C03701=1106.948,-96.023,-47.577,179.847,4.649,148.823
C03702=1106.943,-95.773,-47.587,179.847,4.654,148.825
C03703=1106.938,-95.524,-47.598,179.847,4.660,148.826
C03704=1106.933,-95.274,-47.609,179.846,4.664,148.827
C03705=1106.927,-95.024,-47.619,179.846,4.669,148.828
C03706=1106.922,-94.775,-47.629,179.846,4.674,148.829
C03707=1106.917,-94.525,-47.640,179.845,4.679,148.830
C03708=1106.911,-94.275,-47.650,179.845,4.684,148.832
C03709=1106.907,-94.025,-47.660,179.844,4.689,148.833
C03710=1106.901,-93.776,-47.670,179.844,4.693,148.834
C03711=1106.896,-93.526,-47.680,179.843,4.698,148.835
C03712=1106.891,-93.276,-47.691,179.843,4.703,148.836
C03713=1106.885,-93.027,-47.702,179.842,4.708,148.838
C03714=1106.880,-92.777,-47.713,179.842,4.713,148.839
C03715=1106.875,-92.527,-47.723,179.842,4.718,148.840
C03716=1106.870,-92.277,-47.733,179.841,4.722,148.841
C03717=1106.864,-92.027,-47.744,179.841,4.728,148.842
C03718=1106.859,-91.778,-47.754,179.841,4.733,148.844
C03719=1106.854,-91.528,-47.765,179.840,4.737,148.845
C03720=1106.848,-91.279,-47.775,179.839,4.743,148.846
C03721=1106.843,-91.028,-47.786,179.839,4.748,148.847
C03722=1106.838,-90.779,-47.796,179.839,4.753,148.849
C03723=1106.833,-90.528,-47.807,179.838,4.757,148.850
C03724=1106.827,-90.280,-47.818,179.838,4.762,148.851
C03725=1106.822,-90.029,-47.828,179.838,4.768,148.852
C03726=1106.817,-89.780,-47.838,179.838,4.773,148.853
C03727=1106.812,-89.530,-47.849,179.837,4.777,148.855
C03728=1106.806,-89.281,-47.860,179.837,4.782,148.856
C03729=1106.801,-89.030,-47.870,179.836,4.787,148.857
C03730=1106.796,-88.781,-47.881,179.836,4.793,148.858
C03731=1106.791,-88.531,-47.891,179.835,4.797,148.860
C03732=1106.786,-88.282,-47.902,179.835,4.802,148.861
C03733=1106.781,-88.031,-47.913,179.835,4.807,148.862
C03734=1106.775,-87.782,-47.923,179.834,4.813,148.863
C03735=1106.770,-87.532,-47.934,179.834,4.817,148.864
C03736=1106.765,-87.283,-47.944,179.833,4.822,148.865
C03737=1106.760,-87.069,-47.953,179.833,4.827,148.867
C03738=1106.756,-86.853,-47.963,179.833,4.831,148.868
C03739=1106.752,-86.640,-47.972,179.833,4.835,148.869
C03740=1106.747,-86.424,-47.981,179.832,4.839,148.870
C03741=1106.742,-86.210,-47.991,179.832,4.844,148.871
C03742=1106.738,-85.995,-47.999,179.832,4.849,148.872
C03743=1106.733,-85.781,-48.009,179.831,4.853,148.873
C03744=1106.729,-85.566,-48.017,179.832,4.857,148.874
C03745=1106.724,-85.316,-48.029,179.831,4.862,148.875
C03746=1106.718,-85.067,-48.039,179.830,4.867,148.876
C03747=1106.714,-84.817,-48.050,179.830,4.872,148.877
C03748=1106.708,-84.568,-48.060,179.830,4.877,148.879
C03749=1106.702,-84.317,-48.072,179.830,4.883,148.880
C03750=1106.698,-84.068,-48.083,179.829,4.888,148.881
C03751=1106.692,-83.818,-48.093,179.829,4.893,148.882
C03752=1106.687,-83.568,-48.104,179.829,4.897,148.883
C03753=1106.682,-83.319,-48.115,179.828,4.902,148.885
C03754=1106.677,-83.069,-48.126,179.828,4.907,148.886
C03755=1106.672,-82.820,-48.136,179.828,4.913,148.887
C03756=1106.666,-82.569,-48.147,179.827,4.918,148.888
C03757=1106.661,-82.320,-48.158,179.827,4.923,148.890
C03758=1106.656,-82.070,-48.169,179.827,4.928,148.891
C03759=1106.651,-81.820,-48.180,179.827,4.934,148.892
C03760=1106.645,-81.571,-48.190,179.827,4.939,148.893
C03761=1106.641,-81.321,-48.201,179.827,4.944,148.894
C03762=1106.634,-81.071,-48.212,179.826,4.948,148.895
C03763=1106.629,-80.822,-48.224,179.826,4.953,148.897
C03764=1106.624,-80.571,-48.234,179.825,4.958,148.898
C03765=1106.619,-80.323,-48.245,179.825,4.964,148.899
C03766=1106.615,-80.073,-48.256,179.825,4.969,148.900
C03767=1106.609,-79.822,-48.268,179.824,4.974,148.902
C03768=1106.603,-79.573,-48.278,179.824,4.979,148.903
C03769=1106.598,-79.323,-48.289,179.824,4.985,148.904
C03770=1106.593,-79.074,-48.300,179.824,4.990,148.905
C03771=1106.587,-78.824,-48.311,179.824,4.995,148.906
C03772=1106.583,-78.574,-48.322,179.824,5.000,148.907
C03773=1106.577,-78.325,-48.333,179.823,5.005,148.909
C03774=1106.572,-78.075,-48.344,179.823,5.010,148.910
C03775=1106.567,-77.825,-48.356,179.823,5.015,148.911
C03776=1106.561,-77.575,-48.366,179.823,5.021,148.912
C03777=1106.557,-77.326,-48.377,179.823,5.026,148.913
C03778=1106.551,-77.077,-48.389,179.823,5.031,148.914
C03779=1106.546,-76.826,-48.399,179.823,5.036,148.916
C03780=1106.541,-76.577,-48.411,179.822,5.041,148.917
C03781=1106.535,-76.327,-48.422,179.822,5.046,148.918
C03782=1106.530,-76.077,-48.433,179.822,5.051,148.919
C03783=1106.525,-75.828,-48.444,179.822,5.057,148.920
C03784=1106.520,-75.578,-48.456,179.822,5.062,148.922
C03785=1106.514,-75.328,-48.466,179.822,5.067,148.923
C03786=1106.510,-75.078,-48.477,179.822,5.072,148.924
C03787=1106.504,-74.829,-48.489,179.821,5.077,148.925
C03788=1106.499,-74.580,-48.500,179.821,5.082,148.926
C03789=1106.494,-74.329,-48.511,179.821,5.087,148.927
C03790=1106.488,-74.079,-48.523,179.821,5.093,148.929
C03791=1106.483,-73.831,-48.534,179.821,5.098,148.930
C03792=1106.478,-73.580,-48.544,179.821,5.103,148.931
C03793=1106.474,-73.365,-48.554,179.820,5.107,148.932
C03794=1106.469,-73.151,-48.564,179.821,5.111,148.933
C03795=1106.465,-72.936,-48.574,179.821,5.115,148.934
C03796=1106.460,-72.722,-48.583,179.820,5.121,148.935
C03797=1106.456,-72.508,-48.593,179.820,5.125,148.936
C03798=1106.451,-72.294,-48.603,179.821,5.129,148.937
C03799=1106.447,-72.079,-48.613,179.820,5.133,148.938
C03800=1106.442,-71.865,-48.622,179.820,5.138,148.939
C03801=1106.437,-71.615,-48.633,179.821,5.143,148.940
C03802=1106.432,-71.365,-48.645,179.820,5.148,148.941
C03803=1106.427,-71.115,-48.657,179.820,5.153,148.942
C03804=1106.422,-70.866,-48.668,179.820,5.159,148.943
C03805=1106.416,-70.616,-48.679,179.820,5.164,148.944
C03806=1106.411,-70.366,-48.690,179.820,5.169,148.946
C03807=1106.406,-70.116,-48.702,179.820,5.174,148.947
C03808=1106.401,-69.867,-48.713,179.820,5.179,148.948
C03809=1106.395,-69.617,-48.725,179.820,5.184,148.949
C03810=1106.390,-69.368,-48.736,179.820,5.189,148.950
C03811=1106.385,-69.118,-48.748,179.820,5.194,148.951
C03812=1106.380,-68.868,-48.759,179.820,5.199,148.952
C03813=1106.374,-68.619,-48.771,179.820,5.204,148.953
C03814=1106.370,-68.369,-48.782,179.820,5.209,148.955
C03815=1106.364,-68.119,-48.794,179.820,5.214,148.956
C03816=1106.359,-67.870,-48.805,179.820,5.219,148.957
C03817=1106.354,-67.620,-48.817,179.820,5.224,148.958
C03818=1106.349,-67.370,-48.828,179.820,5.229,148.959
C03819=1106.343,-67.120,-48.839,179.820,5.234,148.960
C03820=1106.338,-66.871,-48.850,179.821,5.240,148.961
C03821=1106.333,-66.621,-48.862,179.821,5.245,148.962
C03822=1106.328,-66.371,-48.874,179.820,5.250,148.963
C03823=1106.323,-66.121,-48.886,179.821,5.255,148.964
C03824=1106.318,-65.872,-48.898,179.821,5.260,148.965
C03825=1106.312,-65.623,-48.909,179.821,5.265,148.966
C03826=1106.307,-65.373,-48.921,179.821,5.270,148.968
C03827=1106.302,-65.123,-48.932,179.821,5.275,148.969
C03828=1106.297,-64.874,-48.944,179.821,5.280,148.970
C03829=1106.292,-64.624,-48.955,179.821,5.285,148.971
C03830=1106.287,-64.374,-48.967,179.821,5.290,148.972
C03831=1106.281,-64.124,-48.979,179.821,5.295,148.973
C03832=1106.277,-63.874,-48.990,179.822,5.300,148.974
C03833=1106.271,-63.625,-49.002,179.822,5.305,148.975
C03834=1106.266,-63.376,-49.013,179.822,5.310,148.976
C03835=1106.260,-63.126,-49.025,179.822,5.315,148.977
C03836=1106.255,-62.876,-49.038,179.823,5.320,148.978
C03837=1106.251,-62.627,-49.049,179.823,5.325,148.979
C03838=1106.245,-62.377,-49.061,179.823,5.330,148.980
C03839=1106.240,-62.127,-49.073,179.823,5.335,148.981
C03840=1106.235,-61.877,-49.084,179.823,5.340,148.982
C03841=1106.230,-61.627,-49.096,179.823,5.345,148.983
C03842=1106.224,-61.378,-49.109,179.824,5.350,148.984
C03843=1106.220,-61.128,-49.120,179.824,5.355,148.985
C03844=1106.214,-60.878,-49.132,179.824,5.360,148.986
C03845=1106.209,-60.628,-49.144,179.824,5.365,148.987
C03846=1106.204,-60.379,-49.155,179.825,5.369,148.988
C03847=1106.199,-60.130,-49.167,179.825,5.374,148.989
C03848=1106.193,-59.880,-49.179,179.825,5.379,148.990
C03849=1106.189,-59.665,-49.189,179.825,5.383,148.991
C03850=1106.185,-59.451,-49.200,179.825,5.388,148.992
C03851=1106.180,-59.237,-49.209,179.825,5.392,148.993
C03852=1106.176,-59.023,-49.220,179.825,5.396,148.994
C03853=1106.171,-58.808,-49.230,179.825,5.400,148.995
C03854=1106.167,-58.594,-49.241,179.824,5.404,148.996
C03855=1106.162,-58.379,-49.250,179.824,5.408,148.997
C03856=1106.158,-58.165,-49.260,179.824,5.412,148.998
C03857=1106.153,-57.915,-49.273,179.824,5.416,148.999
C03858=1106.148,-57.665,-49.285,179.824,5.421,149.000
C03859=1106.143,-57.416,-49.296,179.824,5.425,149.001
C03860=1106.138,-57.166,-49.309,179.824,5.430,149.002
C03861=1106.132,-56.916,-49.321,179.824,5.436,149.003
C03862=1106.127,-56.667,-49.333,179.824,5.440,149.004
C03863=1106.122,-56.418,-49.345,179.824,5.445,149.005
C03864=1106.117,-56.168,-49.357,179.824,5.449,149.006
C03865=1106.112,-55.918,-49.368,179.823,5.454,149.007
C03866=1106.106,-55.668,-49.381,179.823,5.459,149.008
C03867=1106.101,-55.418,-49.393,179.824,5.464,149.009
C03868=1106.097,-55.169,-49.405,179.823,5.468,149.010
C03869=1106.091,-54.919,-49.417,179.823,5.473,149.012
C03870=1106.086,-54.670,-49.429,179.823,5.478,149.013
C03871=1106.081,-54.420,-49.441,179.823,5.482,149.014
C03872=1106.075,-54.170,-49.453,179.823,5.487,149.015
C03873=1106.070,-53.921,-49.466,179.823,5.492,149.016
C03874=1106.065,-53.671,-49.477,179.822,5.496,149.017
C03875=1106.060,-53.422,-49.490,179.823,5.501,149.018
C03876=1106.055,-53.171,-49.502,179.823,5.506,149.019
C03877=1106.050,-52.922,-49.515,179.822,5.511,149.020
C03878=1106.045,-52.672,-49.526,179.822,5.515,149.021
C03879=1106.040,-52.423,-49.539,179.822,5.520,149.022
C03880=1106.034,-52.173,-49.551,179.822,5.525,149.023
C03881=1106.030,-51.923,-49.562,179.822,5.529,149.024
C03882=1106.025,-51.674,-49.575,179.821,5.534,149.025
C03883=1106.019,-51.425,-49.587,179.821,5.539,149.027
C03884=1106.014,-51.175,-49.599,179.822,5.544,149.028
C03885=1106.009,-50.925,-49.612,179.821,5.548,149.029
C03886=1106.003,-50.675,-49.624,179.821,5.553,149.030
C03887=1105.998,-50.426,-49.636,179.821,5.558,149.031
C03888=1105.993,-50.176,-49.648,179.821,5.562,149.032
C03889=1105.988,-49.926,-49.661,179.821,5.567,149.033
C03890=1105.983,-49.676,-49.673,179.821,5.572,149.034
C03891=1105.978,-49.427,-49.686,179.820,5.576,149.035
C03892=1105.972,-49.177,-49.698,179.820,5.581,149.036
C03893=1105.967,-48.928,-49.710,179.821,5.586,149.037
C03894=1105.962,-48.678,-49.723,179.820,5.591,149.038
C03895=1105.957,-48.428,-49.735,179.820,5.596,149.039
C03896=1105.952,-48.179,-49.747,179.819,5.600,149.041
C03897=1105.947,-47.928,-49.760,179.820,5.605,149.042
C03898=1105.942,-47.679,-49.772,179.820,5.610,149.043
C03899=1105.937,-47.430,-49.785,179.819,5.614,149.044
C03900=1105.931,-47.180,-49.797,179.819,5.619,149.045
C03901=1105.926,-46.931,-49.809,179.819,5.624,149.046
C03902=1105.921,-46.681,-49.822,179.819,5.628,149.047
C03903=1105.915,-46.431,-49.834,179.819,5.633,149.048
C03904=1105.911,-46.181,-49.847,179.819,5.638,149.049
C03905=1105.906,-45.968,-49.857,179.819,5.642,149.050
C03906=1105.902,-45.753,-49.868,179.819,5.646,149.051
C03907=1105.898,-45.539,-49.878,179.818,5.650,149.052
C03908=1105.893,-45.324,-49.889,179.818,5.654,149.053
C03909=1105.889,-45.110,-49.900,179.818,5.658,149.054
C03910=1105.884,-44.896,-49.910,179.817,5.662,149.055
C03911=1105.880,-44.682,-49.921,179.817,5.666,149.056
C03912=1105.876,-44.468,-49.932,179.817,5.670,149.057
C03913=1105.870,-44.218,-49.944,179.817,5.675,149.058
C03914=1105.866,-43.968,-49.957,179.817,5.680,149.059
C03915=1105.861,-43.718,-49.970,179.817,5.684,149.060
C03916=1105.855,-43.468,-49.981,179.817,5.689,149.061
C03917=1105.850,-43.219,-49.994,179.817,5.694,149.062
C03918=1105.845,-42.970,-50.007,179.817,5.698,149.063
C03919=1105.840,-42.720,-50.020,179.816,5.704,149.064
C03920=1105.835,-42.470,-50.033,179.817,5.708,149.065
C03921=1105.829,-42.220,-50.045,179.817,5.713,149.066
C03922=1105.824,-41.971,-50.057,179.817,5.718,149.067
C03923=1105.819,-41.721,-50.070,179.818,5.723,149.068
C03924=1105.814,-41.471,-50.083,179.818,5.728,149.069
C03925=1105.809,-41.222,-50.096,179.818,5.733,149.070
C03926=1105.804,-40.972,-50.107,179.819,5.738,149.071
C03927=1105.799,-40.723,-50.120,179.819,5.742,149.072
C03928=1105.793,-40.473,-50.134,179.819,5.747,149.073
C03929=1105.788,-40.223,-50.146,179.819,5.752,149.074
C03930=1105.783,-39.974,-50.159,179.820,5.757,149.075
C03931=1105.778,-39.725,-50.171,179.820,5.762,149.076
C03932=1105.774,-39.475,-50.184,179.821,5.766,149.077
C03933=1105.768,-39.225,-50.197,179.821,5.770,149.078
C03934=1105.762,-38.975,-50.209,179.821,5.775,149.079
C03935=1105.757,-38.726,-50.222,179.821,5.780,149.080
C03936=1105.753,-38.476,-50.235,179.821,5.785,149.081
C03937=1105.747,-38.226,-50.248,179.822,5.790,149.082
C03938=1105.742,-37.977,-50.260,179.822,5.794,149.083
C03939=1105.737,-37.727,-50.274,179.822,5.798,149.083
C03940=1105.732,-37.477,-50.286,179.823,5.803,149.084
C03941=1105.727,-37.228,-50.299,179.823,5.808,149.085
C03942=1105.722,-36.979,-50.312,179.823,5.812,149.086
C03943=1105.716,-36.728,-50.325,179.824,5.817,149.087
C03944=1105.711,-36.479,-50.338,179.824,5.821,149.088
C03945=1105.706,-36.230,-50.350,179.825,5.825,149.089
C03946=1105.702,-35.980,-50.363,179.825,5.830,149.090
C03947=1105.696,-35.730,-50.376,179.826,5.835,149.091
C03948=1105.691,-35.481,-50.389,179.825,5.839,149.091
C03949=1105.686,-35.231,-50.402,179.826,5.844,149.092
C03950=1105.680,-34.981,-50.415,179.826,5.848,149.093
C03951=1105.675,-34.732,-50.428,179.827,5.853,149.094
C03952=1105.671,-34.482,-50.441,179.827,5.857,149.095
C03953=1105.666,-34.233,-50.453,179.827,5.862,149.096
C03954=1105.660,-33.984,-50.467,179.828,5.866,149.097
C03955=1105.655,-33.733,-50.480,179.828,5.870,149.098
C03956=1105.650,-33.484,-50.493,179.828,5.875,149.098
C03957=1105.645,-33.234,-50.506,179.829,5.880,149.099
C03958=1105.640,-32.985,-50.519,179.829,5.883,149.100
C03959=1105.635,-32.735,-50.532,179.829,5.888,149.101
C03960=1105.630,-32.485,-50.545,179.830,5.893,149.102
C03961=1105.626,-32.271,-50.556,179.830,5.896,149.103
C03962=1105.621,-32.057,-50.568,179.830,5.900,149.104
C03963=1105.617,-31.842,-50.579,179.830,5.904,149.104
C03964=1105.612,-31.628,-50.590,179.830,5.907,149.105
C03965=1105.607,-31.413,-50.601,179.831,5.912,149.106
C03966=1105.603,-31.200,-50.612,179.831,5.916,149.107
C03967=1105.598,-30.986,-50.624,179.832,5.919,149.107
C03968=1105.594,-30.772,-50.634,179.831,5.923,149.108
C03969=1105.589,-30.522,-50.649,179.832,5.928,149.109
C03970=1105.584,-30.273,-50.661,179.832,5.932,149.110
C03971=1105.580,-30.023,-50.674,179.832,5.937,149.111
C03972=1105.574,-29.773,-50.687,179.833,5.941,149.112
C03973=1105.569,-29.523,-50.700,179.833,5.945,149.113
C03974=1105.564,-29.274,-50.714,179.833,5.950,149.114
C03975=1105.559,-29.025,-50.727,179.834,5.955,149.115
C03976=1105.554,-28.775,-50.740,179.833,5.959,149.116
C03977=1105.548,-28.525,-50.753,179.834,5.963,149.116
C03978=1105.544,-28.276,-50.767,179.834,5.968,149.117
C03979=1105.538,-28.026,-50.780,179.834,5.972,149.118
C03980=1105.534,-27.776,-50.793,179.835,5.977,149.119
C03981=1105.528,-27.527,-50.807,179.835,5.982,149.120
C03982=1105.524,-27.277,-50.820,179.835,5.985,149.121
C03983=1105.518,-27.027,-50.833,179.835,5.991,149.122
C03984=1105.514,-26.778,-50.847,179.835,5.995,149.123
C03985=1105.508,-26.528,-50.860,179.835,5.999,149.124
C03986=1105.503,-26.278,-50.873,179.836,6.004,149.125
C03987=1105.498,-26.029,-50.887,179.836,6.009,149.126
C03988=1105.493,-25.779,-50.900,179.836,6.014,149.127
C03989=1105.487,-25.530,-50.913,179.836,6.018,149.128
C03990=1105.483,-25.280,-50.927,179.837,6.022,149.129
C03991=1105.477,-25.031,-50.940,179.837,6.028,149.130
C03992=1105.473,-24.781,-50.953,179.837,6.032,149.131
C03993=1105.467,-24.532,-50.967,179.837,6.037,149.132
C03994=1105.463,-24.282,-50.980,179.838,6.042,149.133
C03995=1105.457,-24.033,-50.994,179.838,6.046,149.133
C03996=1105.452,-23.782,-51.007,179.838,6.051,149.135
C03997=1105.447,-23.533,-51.020,179.838,6.056,149.135
C03998=1105.442,-23.283,-51.034,179.839,6.060,149.136
C03999=1105.437,-23.034,-51.047,179.839,6.065,149.137
C04000=1105.432,-22.784,-51.061,179.840,6.070,149.138
C04001=1105.426,-22.535,-51.073,179.840,6.074,149.139
C04002=1105.421,-22.285,-51.088,179.840,6.078,149.140
C04003=1105.416,-22.036,-51.100,179.840,6.083,149.141
C04004=1105.411,-21.786,-51.115,179.841,6.088,149.142
C04005=1105.406,-21.536,-51.128,179.841,6.093,149.143
C04006=1105.401,-21.287,-51.142,179.842,6.098,149.144
C04007=1105.395,-21.037,-51.155,179.841,6.102,149.145
C04008=1105.391,-20.788,-51.169,179.842,6.106,149.146
C04009=1105.386,-20.538,-51.183,179.842,6.111,149.147
C04010=1105.380,-20.289,-51.196,179.843,6.116,149.147
C04011=1105.375,-20.039,-51.210,179.843,6.120,149.148
C04012=1105.370,-19.790,-51.223,179.844,6.125,149.149
C04013=1105.365,-19.540,-51.237,179.844,6.129,149.150
C04014=1105.360,-19.290,-51.251,179.844,6.134,149.151
C04015=1105.355,-19.041,-51.264,179.845,6.139,149.152
C04016=1105.350,-18.791,-51.278,179.845,6.143,149.153
C04017=1105.346,-18.577,-51.289,179.845,6.147,149.154
C04018=1105.341,-18.363,-51.302,179.846,6.152,149.154
C04019=1105.337,-18.149,-51.313,179.846,6.155,149.155
C04020=1105.333,-17.935,-51.324,179.846,6.159,149.156
C04021=1105.328,-17.721,-51.336,179.847,6.163,149.157
C04022=1105.324,-17.507,-51.348,179.847,6.167,149.158
C04023=1105.320,-17.292,-51.361,179.847,6.171,149.158
C04024=1105.315,-17.078,-51.372,179.848,6.174,149.159
C04025=1105.310,-16.829,-51.385,179.848,6.179,149.160
C04026=1105.305,-16.579,-51.400,179.849,6.184,149.161
C04027=1105.300,-16.329,-51.413,179.849,6.189,149.162
C04028=1105.295,-16.080,-51.427,179.850,6.193,149.163
C04029=1105.290,-15.830,-51.441,179.850,6.197,149.163
C04030=1105.285,-15.580,-51.454,179.850,6.202,149.164
C04031=1105.279,-15.331,-51.468,179.851,6.207,149.165
C04032=1105.275,-15.081,-51.483,179.851,6.211,149.166
C04033=1105.270,-14.832,-51.496,179.852,6.216,149.167
C04034=1105.264,-14.582,-51.509,179.853,6.220,149.168
C04035=1105.259,-14.333,-51.524,179.853,6.224,149.169
C04036=1105.255,-14.083,-51.538,179.853,6.229,149.169
C04037=1105.250,-13.834,-51.551,179.854,6.234,149.170
C04038=1105.245,-13.584,-51.566,179.854,6.239,149.171
C04039=1105.239,-13.334,-51.579,179.855,6.243,149.172
C04040=1105.234,-13.085,-51.593,179.856,6.248,149.173
C04041=1105.229,-12.835,-51.607,179.855,6.251,149.174
C04042=1105.224,-12.586,-51.622,179.856,6.256,149.175
C04043=1105.220,-12.336,-51.635,179.856,6.261,149.176
C04044=1105.214,-12.087,-51.649,179.857,6.266,149.176
C04045=1105.209,-11.837,-51.663,179.857,6.270,149.177
C04046=1105.204,-11.587,-51.677,179.858,6.275,149.178
C04047=1105.199,-11.338,-51.691,179.858,6.279,149.179
C04048=1105.194,-11.089,-51.705,179.859,6.283,149.180
C04049=1105.189,-10.839,-51.719,179.859,6.288,149.181
C04050=1105.184,-10.589,-51.733,179.860,6.293,149.182
C04051=1105.179,-10.340,-51.747,179.861,6.297,149.182
C04052=1105.174,-10.091,-51.761,179.861,6.302,149.183
C04053=1105.169,-9.841,-51.776,179.862,6.307,149.184
C04054=1105.164,-9.591,-51.790,179.862,6.310,149.185
C04055=1105.159,-9.342,-51.804,179.862,6.315,149.186
C04056=1105.153,-9.093,-51.818,179.863,6.320,149.187
C04057=1105.148,-8.842,-51.832,179.864,6.324,149.187
C04058=1105.143,-8.593,-51.846,179.864,6.329,149.188
C04059=1105.138,-8.343,-51.860,179.865,6.334,149.189
C04060=1105.133,-8.094,-51.874,179.866,6.338,149.190
C04061=1105.128,-7.844,-51.888,179.866,6.342,149.191
C04062=1105.123,-7.594,-51.903,179.866,6.347,149.192
C04063=1105.118,-7.345,-51.918,179.867,6.351,149.193
C04064=1105.113,-7.096,-51.932,179.868,6.356,149.193
C04065=1105.108,-6.847,-51.946,179.868,6.360,149.194
C04066=1105.103,-6.597,-51.960,179.869,6.365,149.195
C04067=1105.098,-6.347,-51.974,179.869,6.370,149.196
C04068=1105.093,-6.097,-51.989,179.870,6.373,149.197
C04069=1105.088,-5.848,-52.003,179.870,6.378,149.198
C04070=1105.083,-5.598,-52.017,179.871,6.383,149.198
C04071=1105.077,-5.349,-52.031,179.872,6.387,149.199
C04072=1105.072,-5.099,-52.045,179.872,6.392,149.200
C04073=1105.068,-4.885,-52.058,179.873,6.395,149.201
C04074=1105.064,-4.671,-52.070,179.873,6.400,149.202
C04075=1105.060,-4.457,-52.083,179.873,6.404,149.202
C04076=1105.055,-4.243,-52.095,179.874,6.407,149.203
C04077=1105.052,-4.029,-52.107,179.875,6.412,149.204
C04078=1105.047,-3.815,-52.119,179.875,6.415,149.204
C04079=1105.043,-3.601,-52.131,179.875,6.419,149.205
C04080=1105.038,-3.386,-52.144,179.876,6.423,149.206
C04081=1105.033,-3.138,-52.159,179.877,6.428,149.206
C04082=1105.028,-2.888,-52.173,179.877,6.432,149.207
C04083=1105.023,-2.638,-52.187,179.878,6.436,149.208
C04084=1105.018,-2.389,-52.202,179.878,6.441,149.209
C04085=1105.013,-2.139,-52.217,179.879,6.445,149.210
C04086=1105.008,-1.890,-52.231,179.880,6.450,149.211
C04087=1105.003,-1.640,-52.245,179.880,6.455,149.212
C04088=1104.998,-1.390,-52.259,179.881,6.459,149.212
C04089=1104.993,-1.140,-52.274,179.882,6.464,149.213
C04090=1104.987,-0.892,-52.289,179.882,6.468,149.214
C04091=1104.982,-0.642,-52.303,179.883,6.473,149.215
C04092=1104.978,-0.392,-52.317,179.884,6.478,149.216
C04093=1104.973,-0.143,-52.332,179.884,6.481,149.216
C04094=1104.968,0.106,-52.347,179.884,6.486,149.217
C04095=1104.963,0.356,-52.361,179.885,6.490,149.218
C04096=1104.958,0.605,-52.377,179.886,6.495,149.219
C04097=1104.953,0.855,-52.391,179.886,6.500,149.220
C04098=1104.948,1.105,-52.405,179.887,6.504,149.220
C04099=1104.943,1.354,-52.420,179.888,6.509,149.221
C04100=1104.938,1.604,-52.434,179.888,6.514,149.222
C04101=1104.932,1.854,-52.449,179.889,6.518,149.223
C04102=1104.928,2.103,-52.464,179.890,6.523,149.224
C04103=1104.923,2.352,-52.479,179.890,6.527,149.225
C04104=1104.918,2.602,-52.494,179.891,6.532,149.226
C04105=1104.912,2.852,-52.508,179.892,6.536,149.226
C04106=1104.907,3.101,-52.523,179.892,6.541,149.227
C04107=1104.903,3.350,-52.538,179.893,6.546,149.228
C04108=1104.898,3.600,-52.552,179.893,6.551,149.229
C04109=1104.892,3.850,-52.568,179.894,6.555,149.230
C04110=1104.888,4.099,-52.582,179.895,6.560,149.231
C04111=1104.883,4.348,-52.597,179.896,6.564,149.231
C04112=1104.878,4.598,-52.611,179.896,6.569,149.232
C04113=1104.873,4.847,-52.627,179.897,6.573,149.233
C04114=1104.868,5.097,-52.641,179.898,6.578,149.234
C04115=1104.863,5.346,-52.656,179.898,6.583,149.235
C04116=1104.857,5.596,-52.671,179.899,6.587,149.235
C04117=1104.853,5.845,-52.686,179.900,6.592,149.236
C04118=1104.848,6.095,-52.700,179.900,6.596,149.237
C04119=1104.842,6.344,-52.716,179.901,6.601,149.238
C04120=1104.837,6.594,-52.730,179.902,6.606,149.239
C04121=1104.833,6.843,-52.745,179.902,6.610,149.240
C04122=1104.827,7.093,-52.761,179.903,6.615,149.241
C04123=1104.822,7.342,-52.775,179.903,6.620,149.241
C04124=1104.818,7.591,-52.790,179.904,6.624,149.242
C04125=1104.812,7.841,-52.805,179.905,6.629,149.243
C04126=1104.807,8.091,-52.820,179.906,6.633,149.244
C04127=1104.803,8.341,-52.836,179.906,6.638,149.245
C04128=1104.798,8.590,-52.850,179.907,6.643,149.246
C04129=1104.793,8.804,-52.863,179.907,6.646,149.246
C04130=1104.789,9.019,-52.876,179.907,6.650,149.247
C04131=1104.785,9.232,-52.888,179.908,6.655,149.248
C04132=1104.780,9.446,-52.902,179.908,6.658,149.248
C04133=1104.776,9.660,-52.914,179.908,6.662,149.249
C04134=1104.771,9.874,-52.927,179.909,6.666,149.250
C04135=1104.767,10.088,-52.941,179.909,6.669,149.251
C04136=1104.763,10.302,-52.953,179.909,6.673,149.252
C04137=1104.758,10.551,-52.968,179.910,6.678,149.252
C04138=1104.754,10.801,-52.984,179.910,6.682,149.253
C04139=1104.748,11.050,-52.999,179.910,6.686,149.254
C04140=1104.743,11.300,-53.013,179.911,6.691,149.255
C04141=1104.738,11.549,-53.029,179.911,6.696,149.256
C04142=1104.733,11.799,-53.044,179.912,6.700,149.257
C04143=1104.728,12.048,-53.060,179.912,6.704,149.258
C04144=1104.723,12.298,-53.074,179.913,6.709,149.258
C04145=1104.718,12.548,-53.090,179.913,6.713,149.259
C04146=1104.713,12.797,-53.105,179.913,6.717,149.260
C04147=1104.708,13.046,-53.120,179.914,6.722,149.261
C04148=1104.703,13.296,-53.135,179.914,6.727,149.262
C04149=1104.698,13.545,-53.150,179.914,6.731,149.263
C04150=1104.693,13.794,-53.165,179.915,6.735,149.264
C04151=1104.688,14.044,-53.181,179.916,6.740,149.264
C04152=1104.684,14.294,-53.196,179.916,6.743,149.265
C04153=1104.678,14.543,-53.212,179.916,6.748,149.266
C04154=1104.674,14.792,-53.227,179.917,6.753,149.267
C04155=1104.668,15.042,-53.242,179.917,6.756,149.268
C04156=1104.663,15.291,-53.257,179.918,6.761,149.269
C04157=1104.658,15.541,-53.273,179.919,6.766,149.270
C04158=1104.653,15.791,-53.288,179.919,6.771,149.270
C04159=1104.648,16.040,-53.303,179.920,6.774,149.271
C04160=1104.643,16.289,-53.319,179.920,6.779,149.272
C04161=1104.638,16.538,-53.334,179.921,6.783,149.273
C04162=1104.634,16.788,-53.350,179.921,6.787,149.274
C04163=1104.628,17.038,-53.365,179.922,6.792,149.274
C04164=1104.624,17.287,-53.380,179.922,6.796,149.275
C04165=1104.618,17.536,-53.396,179.922,6.800,149.276
C04166=1104.614,17.787,-53.411,179.923,6.805,149.277
C04167=1104.608,18.036,-53.426,179.924,6.809,149.278
C04168=1104.603,18.286,-53.442,179.924,6.813,149.279
C04169=1104.598,18.535,-53.457,179.925,6.818,149.279
C04170=1104.594,18.785,-53.473,179.925,6.822,149.280
C04171=1104.588,19.034,-53.488,179.926,6.826,149.281
C04172=1104.584,19.283,-53.503,179.926,6.830,149.282
C04173=1104.578,19.533,-53.519,179.927,6.835,149.283
C04174=1104.574,19.782,-53.535,179.927,6.839,149.283
C04175=1104.569,20.031,-53.550,179.928,6.843,149.284
C04176=1104.564,20.281,-53.566,179.929,6.848,149.285
C04177=1104.558,20.530,-53.582,179.929,6.852,149.286
C04178=1104.554,20.780,-53.597,179.929,6.856,149.287
C04179=1104.549,21.029,-53.613,179.930,6.861,149.287
C04180=1104.543,21.279,-53.628,179.930,6.865,149.288
C04181=1104.539,21.529,-53.644,179.931,6.869,149.289
C04182=1104.534,21.778,-53.659,179.932,6.874,149.290
C04183=1104.529,22.027,-53.675,179.933,6.878,149.290
C04184=1104.524,22.277,-53.691,179.933,6.882,149.291
C04185=1104.520,22.491,-53.703,179.933,6.885,149.292
C04186=1104.516,22.704,-53.718,179.934,6.889,149.293
C04187=1104.511,22.918,-53.731,179.935,6.893,149.293
C04188=1104.506,23.132,-53.745,179.935,6.897,149.294
C04189=1104.503,23.346,-53.758,179.936,6.900,149.294
C04190=1104.498,23.560,-53.771,179.936,6.904,149.295
C04191=1104.494,23.774,-53.785,179.937,6.907,149.296
C04192=1104.490,23.988,-53.798,179.937,6.911,149.296
C04193=1104.485,24.238,-53.814,179.938,6.915,149.297
C04194=1104.480,24.486,-53.830,179.939,6.920,149.298
C04195=1104.475,24.737,-53.846,179.939,6.923,149.299
C04196=1104.470,24.986,-53.861,179.940,6.928,149.299
C04197=1104.465,25.235,-53.877,179.941,6.932,149.300
C04198=1104.460,25.485,-53.893,179.941,6.936,149.301
C04199=1104.455,25.734,-53.909,179.942,6.940,149.302
C04200=1104.450,25.983,-53.924,179.943,6.945,149.302
C04201=1104.445,26.233,-53.940,179.943,6.948,149.303
C04202=1104.441,26.482,-53.956,179.944,6.953,149.304
C04203=1104.435,26.731,-53.972,179.945,6.957,149.305
C04204=1104.430,26.981,-53.988,179.945,6.961,149.305
C04205=1104.425,27.231,-54.003,179.946,6.966,149.306
C04206=1104.420,27.480,-54.020,179.947,6.970,149.307
C04207=1104.415,27.730,-54.035,179.948,6.974,149.307
C04208=1104.410,27.979,-54.051,179.948,6.978,149.308
C04209=1104.405,28.229,-54.068,179.949,6.982,149.309
C04210=1104.401,28.478,-54.083,179.950,6.987,149.310
C04211=1104.396,28.728,-54.099,179.950,6.991,149.311
C04212=1104.391,28.977,-54.115,179.951,6.995,149.311
C04213=1104.386,29.227,-54.131,179.952,6.999,149.312
C04214=1104.381,29.475,-54.147,179.953,7.003,149.313
C04215=1104.375,29.725,-54.163,179.953,7.007,149.313
C04216=1104.371,29.975,-54.179,179.954,7.012,149.314
C04217=1104.366,30.224,-54.195,179.955,7.015,149.315
C04218=1104.361,30.474,-54.211,179.956,7.020,149.315
C04219=1104.356,30.723,-54.227,179.956,7.024,149.316
C04220=1104.351,30.973,-54.243,179.957,7.028,149.317
C04221=1104.346,31.221,-54.260,179.958,7.032,149.318
C04222=1104.341,31.472,-54.276,179.959,7.036,149.318
C04223=1104.336,31.720,-54.292,179.959,7.040,149.319
C04224=1104.331,31.970,-54.308,179.960,7.045,149.320
C04225=1104.326,32.220,-54.323,179.961,7.049,149.320
C04226=1104.321,32.469,-54.340,179.962,7.052,149.321
C04227=1104.316,32.719,-54.356,179.963,7.057,149.322
C04228=1104.311,32.968,-54.372,179.964,7.061,149.322
C04229=1104.306,33.217,-54.389,179.964,7.065,149.323
C04230=1104.301,33.466,-54.404,179.965,7.069,149.324
C04231=1104.297,33.716,-54.421,179.966,7.074,149.325
C04232=1104.291,33.965,-54.436,179.966,7.077,149.325
C04233=1104.287,34.215,-54.453,179.967,7.081,149.326
C04234=1104.282,34.465,-54.469,179.968,7.086,149.327
C04235=1104.277,34.714,-54.485,179.969,7.090,149.327
C04236=1104.272,34.964,-54.501,179.970,7.093,149.328
C04237=1104.267,35.213,-54.518,179.970,7.098,149.329
C04238=1104.262,35.462,-54.534,179.971,7.102,149.329
C04239=1104.257,35.711,-54.550,179.972,7.106,149.330
C04240=1104.253,35.961,-54.567,179.973,7.110,149.331
C04241=1104.248,36.175,-54.580,179.974,7.113,149.331
C04242=1104.244,36.388,-54.594,179.974,7.117,149.332
C04243=1104.240,36.602,-54.609,179.975,7.120,149.332
C04244=1104.235,36.816,-54.622,179.976,7.124,149.333
C04245=1104.231,37.029,-54.637,179.977,7.128,149.334
C04246=1104.227,37.244,-54.650,179.977,7.131,149.334
C04247=1104.223,37.457,-54.665,179.978,7.135,149.335
C04248=1104.218,37.672,-54.678,179.979,7.138,149.335
C04249=1104.213,37.920,-54.695,179.980,7.142,149.336
C04250=1104.208,38.170,-54.712,179.981,7.147,149.337
C04251=1104.203,38.420,-54.729,179.981,7.150,149.337
C04252=1104.198,38.669,-54.744,179.982,7.154,149.338
C04253=1104.194,38.919,-54.761,179.983,7.159,149.339
C04254=1104.189,39.167,-54.777,179.984,7.162,149.339
C04255=1104.184,39.417,-54.794,179.985,7.167,149.340
C04256=1104.179,39.667,-54.810,179.986,7.171,149.341
C04257=1104.173,39.916,-54.827,179.986,7.174,149.341
C04258=1104.169,40.166,-54.843,179.987,7.179,149.342
C04259=1104.164,40.414,-54.860,179.989,7.183,149.343
C04260=1104.159,40.664,-54.876,179.990,7.187,149.343
C04261=1104.154,40.914,-54.893,179.991,7.190,149.344
C04262=1104.149,41.163,-54.909,179.992,7.195,149.344
C04263=1104.144,41.412,-54.926,179.993,7.199,149.345
C04264=1104.140,41.662,-54.943,179.993,7.203,149.346
C04265=1104.134,41.911,-54.959,179.994,7.207,149.346
C04266=1104.130,42.161,-54.976,179.995,7.211,149.347
C04267=1104.124,42.410,-54.992,179.996,7.215,149.348
C04268=1104.120,42.659,-55.008,179.997,7.219,149.348
C04269=1104.114,42.909,-55.026,179.998,7.223,149.349
C04270=1104.109,43.158,-55.042,179.999,7.228,149.350
C04271=1104.105,43.407,-55.059,180.000,7.231,149.350
C04272=1104.100,43.657,-55.076,-179.999,7.235,149.351
C04273=1104.095,43.906,-55.092,-179.998,7.239,149.351
C04274=1104.090,44.156,-55.109,-179.997,7.243,149.352
C04275=1104.086,44.405,-55.125,-179.996,7.247,149.353
C04276=1104.080,44.655,-55.143,-179.995,7.251,149.353
C04277=1104.075,44.904,-55.159,-179.995,7.255,149.354
C04278=1104.071,45.153,-55.176,-179.993,7.259,149.354
C04279=1104.066,45.403,-55.193,-179.992,7.263,149.355
C04280=1104.061,45.652,-55.209,-179.991,7.267,149.356
C04281=1104.056,45.901,-55.226,-179.991,7.271,149.356
C04282=1104.051,46.151,-55.243,-179.990,7.275,149.357
C04283=1104.046,46.400,-55.260,-179.988,7.279,149.357
C04284=1104.041,46.650,-55.277,-179.988,7.283,149.358
C04285=1104.036,46.899,-55.293,-179.987,7.287,149.359
C04286=1104.032,47.148,-55.310,-179.985,7.291,149.359
C04287=1104.026,47.398,-55.327,-179.984,7.296,149.360
C04288=1104.021,47.647,-55.344,-179.983,7.299,149.360
C04289=1104.016,47.897,-55.361,-179.982,7.303,149.361
C04290=1104.012,48.146,-55.378,-179.981,7.307,149.362
C04291=1104.007,48.396,-55.394,-179.981,7.311,149.362
C04292=1104.002,48.644,-55.412,-179.979,7.315,149.363
C04293=1103.997,48.894,-55.429,-179.978,7.319,149.364
C04294=1103.992,49.144,-55.446,-179.977,7.323,149.364
C04295=1103.987,49.393,-55.463,-179.977,7.327,149.365
C04296=1103.982,49.642,-55.479,-179.975,7.331,149.365
C04297=1103.978,49.856,-55.494,-179.975,7.334,149.366
C04298=1103.974,50.070,-55.508,-179.973,7.338,149.366
C04299=1103.970,50.283,-55.523,-179.972,7.341,149.367
C04300=1103.966,50.497,-55.537,-179.972,7.345,149.367
C04301=1103.961,50.711,-55.552,-179.971,7.348,149.368
C04302=1103.957,50.925,-55.567,-179.970,7.351,149.368
C04303=1103.953,51.138,-55.582,-179.969,7.355,149.369
C04304=1103.949,51.352,-55.597,-179.968,7.358,149.369
C04305=1103.944,51.601,-55.613,-179.967,7.362,149.370
C04306=1103.939,51.851,-55.631,-179.966,7.366,149.371
C04307=1103.934,52.100,-55.647,-179.965,7.370,149.371
C04308=1103.929,52.349,-55.665,-179.964,7.374,149.372
C04309=1103.924,52.598,-55.682,-179.963,7.378,149.372
C04310=1103.919,52.848,-55.699,-179.962,7.382,149.373
C04311=1103.915,53.098,-55.716,-179.960,7.386,149.373
C04312=1103.910,53.347,-55.734,-179.959,7.390,149.374
C04313=1103.905,53.596,-55.750,-179.958,7.394,149.375
C04314=1103.899,53.846,-55.767,-179.957,7.398,149.375
C04315=1103.895,54.095,-55.785,-179.956,7.402,149.376
C04316=1103.890,54.344,-55.802,-179.955,7.406,149.376
C04317=1103.885,54.594,-55.819,-179.954,7.409,149.377
C04318=1103.881,54.843,-55.836,-179.953,7.414,149.377
C04319=1103.875,55.093,-55.854,-179.951,7.417,149.378
C04320=1103.871,55.342,-55.872,-179.950,7.422,149.379
C04321=1103.865,55.591,-55.888,-179.950,7.425,149.379
C04322=1103.860,55.840,-55.905,-179.948,7.429,149.380
C04323=1103.855,56.090,-55.923,-179.947,7.433,149.380
C04324=1103.851,56.339,-55.940,-179.945,7.437,149.381
C04325=1103.846,56.588,-55.958,-179.945,7.441,149.381
C04326=1103.841,56.838,-55.975,-179.944,7.445,149.382
C04327=1103.837,57.087,-55.992,-179.942,7.449,149.383
C04328=1103.831,57.337,-56.010,-179.941,7.453,149.383
C04329=1103.826,57.586,-56.027,-179.940,7.457,149.384
C04330=1103.822,57.835,-56.044,-179.939,7.461,149.384
C04331=1103.817,58.085,-56.062,-179.938,7.465,149.385
C04332=1103.812,58.334,-56.080,-179.936,7.469,149.385
C04333=1103.808,58.583,-56.097,-179.935,7.473,149.386
C04334=1103.802,58.832,-56.114,-179.934,7.476,149.386
C04335=1103.797,59.081,-56.132,-179.933,7.481,149.387
C04336=1103.792,59.331,-56.149,-179.932,7.485,149.388
C04337=1103.788,59.580,-56.167,-179.931,7.489,149.388
C04338=1103.782,59.830,-56.184,-179.930,7.492,149.389
C04339=1103.777,60.079,-56.202,-179.929,7.496,149.389
C04340=1103.773,60.329,-56.218,-179.927,7.500,149.390
C04341=1103.768,60.578,-56.236,-179.926,7.504,149.390
C04342=1103.763,60.827,-56.254,-179.924,7.508,149.391
C04343=1103.758,61.077,-56.272,-179.924,7.512,149.391
C04344=1103.753,61.326,-56.290,-179.922,7.516,149.392
C04345=1103.749,61.575,-56.307,-179.921,7.520,149.393
C04346=1103.744,61.825,-56.324,-179.920,7.524,149.393
C04347=1103.739,62.074,-56.342,-179.919,7.528,149.394
C04348=1103.734,62.323,-56.360,-179.918,7.531,149.394
C04349=1103.729,62.573,-56.378,-179.916,7.535,149.394
C04350=1103.724,62.822,-56.395,-179.915,7.540,149.395
C04351=1103.719,63.071,-56.413,-179.913,7.543,149.396
C04352=1103.714,63.321,-56.430,-179.912,7.548,149.396
C04353=1103.710,63.535,-56.446,-179.911,7.551,149.397
C04354=1103.706,63.748,-56.461,-179.910,7.554,149.397
C04355=1103.702,63.962,-56.476,-179.909,7.557,149.398
C04356=1103.698,64.175,-56.491,-179.908,7.561,149.398
C04357=1103.694,64.389,-56.507,-179.907,7.564,149.398
C04358=1103.690,64.602,-56.522,-179.906,7.567,149.399
C04359=1103.685,64.816,-56.537,-179.906,7.571,149.400
C04360=1103.681,65.029,-56.552,-179.904,7.575,149.400
C04361=1103.677,65.279,-56.570,-179.902,7.579,149.400
C04362=1103.672,65.529,-56.587,-179.901,7.582,149.401
C04363=1103.667,65.778,-56.605,-179.900,7.586,149.401
C04364=1103.662,66.027,-56.623,-179.899,7.590,149.402
C04365=1103.657,66.276,-56.641,-179.898,7.594,149.403
C04366=1103.652,66.525,-56.659,-179.896,7.598,149.403
C04367=1103.647,66.774,-56.677,-179.895,7.601,149.403
C04368=1103.642,67.024,-56.695,-179.894,7.606,149.404
C04369=1103.637,67.273,-56.713,-179.892,7.609,149.405
C04370=1103.632,67.523,-56.731,-179.891,7.614,149.405
C04371=1103.628,67.773,-56.749,-179.890,7.618,149.406
C04372=1103.623,68.022,-56.767,-179.888,7.622,149.406
C04373=1103.618,68.271,-56.785,-179.888,7.625,149.407
C04374=1103.613,68.520,-56.803,-179.886,7.629,149.407
C04375=1103.608,68.769,-56.821,-179.885,7.633,149.408
C04376=1103.603,69.018,-56.839,-179.883,7.637,149.408
C04377=1103.599,69.268,-56.857,-179.882,7.641,149.409
C04378=1103.594,69.517,-56.875,-179.881,7.645,149.409
C04379=1103.589,69.767,-56.893,-179.879,7.649,149.410
C04380=1103.584,70.016,-56.911,-179.878,7.652,149.410
C04381=1103.580,70.265,-56.929,-179.877,7.657,149.411
C04382=1103.575,70.514,-56.947,-179.876,7.660,149.411
C04383=1103.570,70.763,-56.965,-179.874,7.664,149.412
C04384=1103.565,71.013,-56.983,-179.873,7.669,149.412
C04385=1103.560,71.262,-57.001,-179.871,7.673,149.413
C04386=1103.556,71.512,-57.019,-179.870,7.676,149.413
C04387=1103.551,71.761,-57.037,-179.869,7.680,149.414
C04388=1103.546,72.010,-57.055,-179.868,7.684,149.414
C04389=1103.541,72.259,-57.073,-179.866,7.688,149.415
C04390=1103.537,72.509,-57.092,-179.865,7.692,149.415
C04391=1103.531,72.758,-57.110,-179.863,7.696,149.416
C04392=1103.526,73.008,-57.128,-179.862,7.700,149.416
C04393=1103.521,73.256,-57.147,-179.861,7.704,149.417
C04394=1103.517,73.506,-57.165,-179.859,7.708,149.417
C04395=1103.512,73.755,-57.183,-179.858,7.711,149.418
C04396=1103.507,74.004,-57.201,-179.857,7.715,149.418
C04397=1103.502,74.254,-57.219,-179.856,7.719,149.419
C04398=1103.498,74.503,-57.238,-179.854,7.723,149.419
C04399=1103.493,74.752,-57.257,-179.853,7.728,149.420
C04400=1103.488,75.002,-57.275,-179.851,7.731,149.420
C04401=1103.483,75.251,-57.293,-179.850,7.735,149.421
C04402=1103.479,75.501,-57.311,-179.849,7.740,149.422
C04403=1103.474,75.749,-57.330,-179.847,7.743,149.422
C04404=1103.468,75.999,-57.348,-179.846,7.747,149.422
C04405=1103.463,76.248,-57.366,-179.844,7.751,149.423
C04406=1103.459,76.498,-57.385,-179.843,7.755,149.423
C04407=1103.454,76.746,-57.403,-179.842,7.759,149.424
C04408=1103.449,76.996,-57.422,-179.840,7.763,149.424
C04409=1103.446,77.209,-57.438,-179.839,7.766,149.425
C04410=1103.441,77.423,-57.453,-179.839,7.769,149.425
C04411=1103.437,77.636,-57.469,-179.838,7.772,149.426
C04412=1103.433,77.850,-57.485,-179.837,7.775,149.426
C04413=1103.429,78.064,-57.501,-179.836,7.779,149.427
C04414=1103.424,78.277,-57.517,-179.835,7.782,149.427
C04415=1103.420,78.491,-57.532,-179.834,7.785,149.428
C04416=1103.416,78.704,-57.549,-179.833,7.788,149.428
C04417=1103.411,78.953,-57.567,-179.832,7.791,149.429
C04418=1103.406,79.202,-57.585,-179.831,7.796,149.429
C04419=1103.402,79.452,-57.605,-179.831,7.799,149.430
C04420=1103.397,79.701,-57.623,-179.829,7.803,149.430
C04421=1103.392,79.950,-57.641,-179.829,7.807,149.431
C04422=1103.387,80.200,-57.660,-179.827,7.810,149.432
C04423=1103.382,80.449,-57.678,-179.827,7.814,149.432
C04424=1103.378,80.698,-57.697,-179.825,7.818,149.433
C04425=1103.373,80.948,-57.716,-179.825,7.821,149.433
C04426=1103.368,81.196,-57.735,-179.823,7.825,149.434
C04427=1103.364,81.446,-57.753,-179.822,7.829,149.434
C04428=1103.358,81.695,-57.772,-179.821,7.833,149.435
C04429=1103.353,81.944,-57.790,-179.820,7.836,149.435
C04430=1103.349,82.193,-57.809,-179.819,7.840,149.436
C04431=1103.344,82.443,-57.828,-179.818,7.844,149.437
C04432=1103.340,82.692,-57.847,-179.817,7.848,149.437
C04433=1103.335,82.941,-57.865,-179.816,7.852,149.438
C04434=1103.329,83.190,-57.884,-179.815,7.855,149.438
C04435=1103.325,83.440,-57.903,-179.813,7.859,149.439
C04436=1103.320,83.689,-57.922,-179.813,7.863,149.439
C04437=1103.316,83.939,-57.940,-179.811,7.866,149.440
C04438=1103.311,84.187,-57.959,-179.810,7.870,149.440
C04439=1103.305,84.437,-57.977,-179.809,7.874,149.441
C04440=1103.301,84.686,-57.997,-179.808,7.878,149.441
C04441=1103.296,84.935,-58.016,-179.807,7.881,149.442
C04442=1103.292,85.185,-58.034,-179.806,7.885,149.442
C04443=1103.286,85.434,-58.053,-179.805,7.889,149.443
C04444=1103.282,85.684,-58.072,-179.804,7.892,149.443
C04445=1103.277,85.933,-58.091,-179.802,7.897,149.444
C04446=1103.272,86.181,-58.110,-179.801,7.900,149.445
C04447=1103.267,86.431,-58.129,-179.800,7.904,149.445
C04448=1103.262,86.680,-58.147,-179.799,7.907,149.446
C04449=1103.258,86.929,-58.167,-179.798,7.911,149.446
C04450=1103.253,87.179,-58.185,-179.797,7.915,149.447
C04451=1103.248,87.428,-58.205,-179.796,7.919,149.447
C04452=1103.243,87.677,-58.223,-179.794,7.923,149.448
C04453=1103.239,87.926,-58.243,-179.794,7.926,149.448
C04454=1103.234,88.175,-58.261,-179.792,7.930,149.449
C04455=1103.229,88.425,-58.281,-179.791,7.934,149.449
C04456=1103.224,88.674,-58.299,-179.790,7.937,149.450
C04457=1103.220,88.923,-58.319,-179.789,7.941,149.450
C04458=1103.215,89.172,-58.337,-179.787,7.945,149.451
C04459=1103.210,89.422,-58.357,-179.786,7.948,149.451
C04460=1103.205,89.670,-58.375,-179.785,7.953,149.452
C04461=1103.201,89.920,-58.395,-179.783,7.957,149.452
C04462=1103.195,90.170,-58.414,-179.782,7.960,149.453
C04463=1103.191,90.419,-58.433,-179.781,7.964,149.453
C04464=1103.186,90.668,-58.452,-179.780,7.968,149.454
C04465=1103.179,91.057,-58.482,-179.778,7.973,149.455
C04466=1103.171,91.446,-58.512,-179.776,7.979,149.455
C04467=1103.164,91.835,-58.542,-179.774,7.985,149.456
C04468=1103.156,92.225,-58.572,-179.772,7.991,149.457
C04469=1103.152,92.473,-58.591,-179.771,7.995,149.458
C04470=1103.147,92.724,-58.610,-179.770,7.999,149.458
C04471=1103.141,92.973,-58.629,-179.768,8.002,149.458
C04472=1103.137,93.222,-58.648,-179.767,8.006,149.459
C04473=1102.909,83.212,-57.935,-179.811,7.858,149.438
C04474=1102.913,82.964,-57.916,-179.812,7.854,149.437
C04475=1102.918,82.713,-57.897,-179.813,7.851,149.437
C04476=1102.923,82.465,-57.878,-179.814,7.846,149.436
C04477=1102.927,82.215,-57.860,-179.815,7.843,149.435
C04478=1102.933,81.966,-57.841,-179.816,7.839,149.435
C04479=1102.938,81.717,-57.823,-179.817,7.836,149.434
C04480=1102.942,81.468,-57.804,-179.818,7.831,149.434
C04481=1102.947,81.218,-57.785,-179.820,7.828,149.433
C04482=1102.952,80.970,-57.766,-179.820,7.824,149.433
C04483=1102.957,80.719,-57.748,-179.822,7.820,149.432
C04484=1102.961,80.471,-57.729,-179.822,7.817,149.432
C04485=1102.966,80.221,-57.710,-179.824,7.813,149.431
C04486=1102.971,79.971,-57.692,-179.824,7.809,149.430
C04487=1102.976,79.723,-57.673,-179.825,7.805,149.430
C04488=1102.980,79.473,-57.655,-179.826,7.802,149.429
C04489=1102.985,79.225,-57.636,-179.827,7.798,149.429
C04490=1102.991,78.975,-57.618,-179.828,7.795,149.428
C04491=1102.995,78.725,-57.599,-179.830,7.790,149.428
C04492=1103.000,78.477,-57.581,-179.831,7.787,149.427
C04493=1103.005,78.227,-57.562,-179.832,7.783,149.427
C04494=1103.011,77.921,-57.540,-179.833,7.779,149.426
C04495=1103.016,77.615,-57.516,-179.834,7.774,149.425
C04496=1103.023,77.308,-57.493,-179.835,7.770,149.425
C04497=1103.028,77.001,-57.471,-179.836,7.765,149.424
C04498=1103.034,76.752,-57.452,-179.837,7.761,149.423
C04499=1103.038,76.503,-57.434,-179.839,7.758,149.423
C04500=1103.043,76.254,-57.415,-179.840,7.754,149.422
C04501=1103.048,76.004,-57.397,-179.842,7.749,149.422
C04502=1103.052,75.755,-57.379,-179.843,7.745,149.421
C04503=1103.057,75.506,-57.360,-179.845,7.742,149.421
C04504=1103.062,75.256,-57.342,-179.846,7.737,149.420
C04505=1103.067,75.007,-57.324,-179.847,7.733,149.420
C04506=1103.072,74.758,-57.306,-179.849,7.730,149.419
C04507=1103.076,74.509,-57.287,-179.850,7.725,149.419
C04508=1103.082,74.259,-57.268,-179.851,7.722,149.418
C04509=1103.086,74.010,-57.250,-179.853,7.718,149.418
C04510=1103.091,73.761,-57.232,-179.854,7.714,149.417
C04511=1103.096,73.511,-57.214,-179.855,7.710,149.417
C04512=1103.101,73.262,-57.196,-179.857,7.706,149.416
C04513=1103.105,73.013,-57.177,-179.858,7.702,149.416
C04514=1103.110,72.764,-57.159,-179.860,7.698,149.415
C04515=1103.115,72.514,-57.140,-179.861,7.694,149.415
C04516=1103.120,72.265,-57.122,-179.862,7.691,149.414
C04517=1103.125,72.016,-57.104,-179.863,7.687,149.414
C04518=1103.130,71.767,-57.086,-179.865,7.683,149.413
C04519=1103.135,71.517,-57.068,-179.866,7.679,149.413
C04520=1103.139,71.267,-57.050,-179.868,7.675,149.412
C04521=1103.144,71.018,-57.032,-179.869,7.671,149.412
C04522=1103.149,70.769,-57.014,-179.871,7.667,149.411
C04523=1103.154,70.521,-56.995,-179.871,7.663,149.411
C04524=1103.158,70.271,-56.977,-179.873,7.659,149.410
C04525=1103.163,70.022,-56.959,-179.874,7.655,149.410
C04526=1103.168,69.772,-56.941,-179.875,7.651,149.409
C04527=1103.173,69.523,-56.923,-179.877,7.647,149.409
C04528=1103.178,69.274,-56.905,-179.878,7.643,149.408
C04529=1103.183,69.024,-56.887,-179.880,7.639,149.408
C04530=1103.188,68.775,-56.869,-179.881,7.636,149.407
C04531=1103.193,68.526,-56.851,-179.882,7.632,149.406
C04532=1103.198,68.276,-56.833,-179.883,7.628,149.406
C04533=1103.203,68.026,-56.815,-179.885,7.624,149.406
C04534=1103.207,67.777,-56.797,-179.886,7.620,149.405
C04535=1103.212,67.528,-56.779,-179.888,7.616,149.405
C04536=1103.217,67.279,-56.762,-179.888,7.612,149.404
C04537=1103.221,67.030,-56.744,-179.890,7.608,149.403
C04538=1103.226,66.781,-56.726,-179.891,7.604,149.403
C04539=1103.231,66.532,-56.708,-179.892,7.600,149.402
C04540=1103.236,66.282,-56.689,-179.894,7.596,149.402
C04541=1103.240,66.033,-56.671,-179.895,7.592,149.401
C04542=1103.246,65.783,-56.654,-179.896,7.589,149.401
C04543=1103.251,65.534,-56.636,-179.897,7.585,149.400
C04544=1103.256,65.285,-56.618,-179.899,7.581,149.400
C04545=1103.260,65.035,-56.600,-179.900,7.577,149.399
C04546=1103.264,64.822,-56.586,-179.901,7.574,149.399
C04547=1103.269,64.608,-56.570,-179.902,7.570,149.398
C04548=1103.273,64.395,-56.554,-179.903,7.566,149.398
C04549=1103.277,64.180,-56.539,-179.904,7.563,149.397
C04550=1103.281,63.967,-56.524,-179.905,7.560,149.397
C04551=1103.285,63.753,-56.509,-179.906,7.557,149.396
C04552=1103.289,63.540,-56.494,-179.908,7.553,149.396
C04553=1103.293,63.326,-56.479,-179.908,7.550,149.396
C04554=1103.298,63.077,-56.461,-179.910,7.545,149.395
C04555=1103.303,62.828,-56.443,-179.911,7.542,149.395
C04556=1103.308,62.579,-56.425,-179.912,7.538,149.394
C04557=1103.313,62.329,-56.408,-179.913,7.534,149.393
C04558=1103.318,62.080,-56.391,-179.915,7.530,149.393
C04559=1103.323,61.831,-56.373,-179.916,7.526,149.392
C04560=1103.328,61.581,-56.355,-179.917,7.522,149.392
C04561=1103.333,61.332,-56.337,-179.918,7.519,149.391
C04562=1103.338,61.083,-56.319,-179.919,7.515,149.391
C04563=1103.342,60.833,-56.303,-179.921,7.510,149.390
C04564=1103.347,60.584,-56.285,-179.922,7.506,149.390
C04565=1103.352,60.335,-56.267,-179.923,7.503,149.389
C04566=1103.357,60.085,-56.249,-179.924,7.499,149.389
C04567=1103.362,59.836,-56.232,-179.925,7.495,149.388
C04568=1103.366,59.586,-56.215,-179.927,7.491,149.388
C04569=1103.371,59.337,-56.197,-179.928,7.487,149.387
C04570=1103.376,59.088,-56.179,-179.929,7.483,149.386
C04571=1103.381,58.839,-56.162,-179.930,7.479,149.386
C04572=1103.386,58.589,-56.144,-179.931,7.475,149.385
C04573=1103.391,58.340,-56.127,-179.933,7.471,149.385
C04574=1103.396,58.091,-56.109,-179.933,7.467,149.384
C04575=1103.400,57.841,-56.092,-179.935,7.464,149.384
C04576=1103.405,57.592,-56.074,-179.936,7.459,149.383
C04577=1103.410,57.342,-56.057,-179.937,7.455,149.383
C04578=1103.415,57.093,-56.040,-179.938,7.452,149.382
C04579=1103.420,56.843,-56.022,-179.939,7.448,149.381
C04580=1103.425,56.594,-56.004,-179.940,7.444,149.381
C04581=1103.430,56.345,-55.988,-179.942,7.439,149.380
C04582=1103.435,56.096,-55.970,-179.943,7.435,149.380
C04583=1103.440,55.846,-55.953,-179.944,7.432,149.379
C04584=1103.444,55.597,-55.936,-179.945,7.428,149.379
C04585=1103.449,55.348,-55.918,-179.946,7.424,149.378
C04586=1103.455,55.098,-55.901,-179.947,7.419,149.377
C04587=1103.459,54.849,-55.884,-179.948,7.416,149.377
C04588=1103.464,54.599,-55.866,-179.949,7.412,149.376
C04589=1103.468,54.350,-55.850,-179.951,7.408,149.376
C04590=1103.474,54.101,-55.832,-179.952,7.404,149.375
C04591=1103.479,53.852,-55.815,-179.952,7.400,149.374
C04592=1103.484,53.602,-55.798,-179.954,7.396,149.374
C04593=1103.489,53.353,-55.780,-179.955,7.392,149.373
C04594=1103.493,53.103,-55.763,-179.956,7.389,149.373
C04595=1103.498,52.854,-55.746,-179.957,7.385,149.372
C04596=1103.503,52.604,-55.728,-179.958,7.380,149.372
C04597=1103.508,52.356,-55.712,-179.959,7.376,149.371
C04598=1103.513,52.106,-55.695,-179.960,7.373,149.371
C04599=1103.518,51.857,-55.677,-179.961,7.369,149.370
C04600=1103.523,51.607,-55.660,-179.962,7.364,149.369
C04601=1103.527,51.358,-55.643,-179.964,7.360,149.369
C04602=1103.532,51.144,-55.628,-179.964,7.357,149.368
C04603=1103.536,50.930,-55.614,-179.965,7.354,149.368
C04604=1103.540,50.716,-55.599,-179.966,7.351,149.367
C04605=1103.545,50.503,-55.585,-179.967,7.348,149.367
C04606=1103.549,50.289,-55.570,-179.968,7.343,149.366
C04607=1103.553,50.076,-55.555,-179.969,7.340,149.366
C04608=1103.557,49.863,-55.541,-179.970,7.337,149.365
C04609=1103.561,49.649,-55.526,-179.971,7.334,149.365
C04610=1103.566,49.399,-55.509,-179.972,7.329,149.364
C04611=1103.571,49.150,-55.492,-179.973,7.325,149.364
C04612=1103.576,48.900,-55.475,-179.974,7.322,149.363
C04613=1103.581,48.651,-55.459,-179.975,7.318,149.362
C04614=1103.586,48.401,-55.442,-179.976,7.314,149.362
C04615=1103.590,48.152,-55.424,-179.977,7.309,149.361
C04616=1103.595,47.903,-55.408,-179.978,7.306,149.360
C04617=1103.601,47.654,-55.391,-179.979,7.301,149.360
C04618=1103.605,47.404,-55.374,-179.980,7.297,149.359
C04619=1103.610,47.154,-55.357,-179.981,7.294,149.359
C04620=1103.615,46.905,-55.340,-179.982,7.290,149.358
C04621=1103.620,46.656,-55.324,-179.983,7.285,149.357
C04622=1103.625,46.406,-55.307,-179.984,7.281,149.357
C04623=1103.630,46.157,-55.290,-179.985,7.278,149.356
C04624=1103.635,45.907,-55.273,-179.986,7.274,149.356
C04625=1103.640,45.658,-55.256,-179.987,7.269,149.355
C04626=1103.644,45.409,-55.240,-179.988,7.266,149.354
C04627=1103.650,45.159,-55.222,-179.989,7.262,149.354
C04628=1103.654,44.910,-55.206,-179.990,7.257,149.353
C04629=1103.659,44.661,-55.189,-179.991,7.254,149.353
C04630=1103.664,44.411,-55.172,-179.992,7.250,149.352
C04631=1103.669,44.162,-55.155,-179.993,7.246,149.351
C04632=1103.674,43.913,-55.139,-179.994,7.241,149.351
C04633=1103.679,43.663,-55.122,-179.995,7.238,149.350
C04634=1103.684,43.413,-55.105,-179.996,7.233,149.349
C04635=1103.689,43.165,-55.089,-179.997,7.229,149.349
C04636=1103.693,42.915,-55.072,-179.998,7.226,149.348
C04637=1103.698,42.665,-55.055,-179.999,7.222,149.348
C04638=1103.704,42.417,-55.039,-180.000,7.217,149.347
C04639=1103.708,42.167,-55.022,180.000,7.214,149.346
C04640=1103.713,41.917,-55.005,179.999,7.210,149.346
C04641=1103.718,41.669,-54.988,179.998,7.205,149.345
C04642=1103.723,41.418,-54.972,179.997,7.201,149.344
C04643=1103.728,41.169,-54.956,179.996,7.198,149.344
C04644=1103.733,40.920,-54.939,179.995,7.193,149.343
C04645=1103.738,40.670,-54.922,179.994,7.189,149.342
C04646=1103.742,40.421,-54.906,179.993,7.185,149.342
C04647=1103.747,40.172,-54.889,179.992,7.181,149.341
C04648=1103.753,39.922,-54.873,179.991,7.177,149.340
C04649=1103.757,39.672,-54.856,179.991,7.173,149.340
C04650=1103.763,39.423,-54.840,179.990,7.169,149.339
C04651=1103.767,39.174,-54.823,179.989,7.165,149.338
C04652=1103.772,38.925,-54.807,179.988,7.162,149.338
C04653=1103.777,38.675,-54.791,179.987,7.157,149.337
C04654=1103.782,38.425,-54.774,179.986,7.153,149.337
C04655=1103.787,38.177,-54.757,179.986,7.149,149.336
C04656=1103.792,37.927,-54.741,179.985,7.145,149.335
C04657=1103.797,37.678,-54.725,179.984,7.140,149.334
C04658=1103.801,37.464,-54.711,179.983,7.137,149.334
C04659=1103.805,37.250,-54.697,179.982,7.134,149.333
C04660=1103.809,37.036,-54.682,179.981,7.131,149.333
C04661=1103.814,36.823,-54.668,179.981,7.127,149.332
C04662=1103.818,36.609,-54.655,179.980,7.123,149.332
C04663=1103.822,36.395,-54.640,179.979,7.120,149.331
C04664=1103.826,36.181,-54.627,179.978,7.116,149.331
C04665=1103.831,35.968,-54.612,179.977,7.113,149.330
C04666=1103.836,35.718,-54.596,179.977,7.108,149.329
C04667=1103.841,35.469,-54.580,179.976,7.105,149.329
C04668=1103.845,35.219,-54.564,179.975,7.101,149.328
C04669=1103.850,34.970,-54.547,179.974,7.096,149.327
C04670=1103.855,34.720,-54.531,179.974,7.093,149.327
C04671=1103.860,34.471,-54.514,179.973,7.088,149.326
C04672=1103.866,34.221,-54.498,179.972,7.084,149.325
C04673=1103.870,33.972,-54.482,179.971,7.080,149.325
C04674=1103.876,33.722,-54.466,179.970,7.076,149.324
C04675=1103.880,33.473,-54.450,179.970,7.072,149.323
C04676=1103.885,33.224,-54.433,179.969,7.067,149.322
C04677=1103.890,32.974,-54.417,179.968,7.064,149.322
C04678=1103.895,32.725,-54.401,179.967,7.059,149.321
C04679=1103.900,32.475,-54.385,179.966,7.055,149.320
C04680=1103.905,32.226,-54.369,179.966,7.052,149.320
C04681=1103.910,31.976,-54.353,179.965,7.047,149.319
C04682=1103.915,31.727,-54.336,179.964,7.043,149.318
C04683=1103.920,31.477,-54.321,179.963,7.039,149.318
C04684=1103.925,31.228,-54.304,179.962,7.035,149.317
C04685=1103.930,30.978,-54.288,179.961,7.031,149.316
C04686=1103.935,30.730,-54.272,179.961,7.027,149.315
C04687=1103.940,30.480,-54.256,179.960,7.022,149.315
C04688=1103.944,30.231,-54.240,179.959,7.018,149.314
C04689=1103.950,29.981,-54.224,179.959,7.014,149.313
C04690=1103.955,29.731,-54.208,179.958,7.010,149.313
C04691=1103.960,29.482,-54.192,179.957,7.005,149.312
C04692=1103.965,29.232,-54.176,179.957,7.002,149.311
C04693=1103.969,28.984,-54.160,179.956,6.997,149.310
C04694=1103.974,28.734,-54.144,179.955,6.993,149.310
C04695=1103.979,28.484,-54.129,179.955,6.989,149.309
C04696=1103.984,28.236,-54.112,179.954,6.985,149.308
C04697=1103.989,27.985,-54.096,179.953,6.980,149.307
C04698=1103.994,27.736,-54.081,179.953,6.977,149.307
C04699=1103.999,27.487,-54.064,179.951,6.973,149.306
C04700=1104.004,27.237,-54.049,179.951,6.968,149.305
C04701=1104.010,26.988,-54.033,179.950,6.964,149.305
C04702=1104.014,26.738,-54.016,179.949,6.960,149.304
C04703=1104.019,26.489,-54.001,179.949,6.955,149.303
C04704=1104.023,26.239,-53.985,179.948,6.952,149.302
C04705=1104.029,25.990,-53.969,179.948,6.947,149.302
C04706=1104.034,25.741,-53.953,179.947,6.943,149.301
C04707=1104.039,25.491,-53.937,179.946,6.939,149.300
C04708=1104.044,25.242,-53.921,179.946,6.935,149.299
C04709=1104.048,24.992,-53.906,179.945,6.930,149.299
C04710=1104.053,24.743,-53.890,179.945,6.926,149.298
C04711=1104.059,24.493,-53.875,179.944,6.922,149.297
C04712=1104.063,24.243,-53.859,179.943,6.918,149.296
C04713=1104.068,23.994,-53.842,179.943,6.914,149.296
C04714=1104.072,23.780,-53.829,179.942,6.910,149.295
C04715=1104.077,23.567,-53.816,179.941,6.906,149.294
C04716=1104.081,23.353,-53.802,179.941,6.903,149.294
C04717=1104.086,23.139,-53.789,179.940,6.899,149.293
C04718=1104.090,22.925,-53.776,179.940,6.896,149.292
C04719=1104.094,22.711,-53.762,179.939,6.892,149.292
C04720=1104.099,22.498,-53.748,179.939,6.888,149.291
C04721=1104.102,22.284,-53.735,179.939,6.885,149.290
C04722=1104.108,22.034,-53.719,179.938,6.881,149.290
C04723=1104.113,21.785,-53.704,179.937,6.876,149.289
C04724=1104.117,21.535,-53.688,179.937,6.872,149.288
C04725=1104.122,21.286,-53.673,179.936,6.868,149.287
C04726=1104.128,21.036,-53.657,179.935,6.863,149.287
C04727=1104.133,20.786,-53.641,179.935,6.860,149.286
C04728=1104.137,20.538,-53.626,179.934,6.855,149.285
C04729=1104.142,20.288,-53.610,179.933,6.850,149.284
C04730=1104.147,20.038,-53.594,179.933,6.847,149.283
C04731=1104.152,19.789,-53.579,179.932,6.842,149.283
C04732=1104.157,19.540,-53.563,179.932,6.838,149.282
C04733=1104.162,19.290,-53.548,179.932,6.834,149.281
C04734=1104.166,19.040,-53.532,179.931,6.829,149.280
C04735=1104.172,18.791,-53.517,179.930,6.825,149.279
C04736=1104.177,18.542,-53.501,179.930,6.821,149.279
C04737=1104.182,18.293,-53.486,179.929,6.816,149.278
C04738=1104.187,18.042,-53.470,179.929,6.812,149.277
C04739=1104.192,17.793,-53.455,179.928,6.808,149.276
C04740=1104.197,17.544,-53.440,179.928,6.804,149.275
C04741=1104.202,17.295,-53.424,179.927,6.799,149.274
C04742=1104.207,17.044,-53.408,179.927,6.795,149.274
C04743=1104.212,16.795,-53.393,179.926,6.791,149.273
C04744=1104.217,16.546,-53.378,179.926,6.786,149.272
C04745=1104.222,16.297,-53.362,179.925,6.781,149.271
C04746=1104.226,16.047,-53.347,179.925,6.778,149.270
C04747=1104.232,15.797,-53.331,179.924,6.773,149.270
C04748=1104.237,15.548,-53.317,179.923,6.768,149.269
C04749=1104.242,15.298,-53.301,179.924,6.764,149.268
C04750=1104.247,15.049,-53.286,179.922,6.760,149.267
C04751=1104.252,14.799,-53.270,179.922,6.755,149.266
C04752=1104.257,14.550,-53.255,179.922,6.751,149.265
C04753=1104.262,14.301,-53.240,179.921,6.747,149.264
C04754=1104.267,14.051,-53.224,179.921,6.742,149.264
C04755=1104.272,13.802,-53.209,179.920,6.738,149.263
C04756=1104.277,13.551,-53.194,179.920,6.734,149.262
C04757=1104.281,13.302,-53.179,179.919,6.729,149.261
C04758=1104.287,13.053,-53.163,179.919,6.725,149.260
C04759=1104.291,12.804,-53.148,179.919,6.720,149.259
C04760=1104.297,12.554,-53.133,179.918,6.716,149.258
C04761=1104.301,12.305,-53.118,179.918,6.712,149.258
C04762=1104.307,12.054,-53.103,179.917,6.708,149.257
C04763=1104.311,11.805,-53.088,179.917,6.703,149.256
C04764=1104.317,11.556,-53.072,179.917,6.699,149.255
C04765=1104.321,11.307,-53.057,179.916,6.694,149.254
C04766=1104.327,11.057,-53.042,179.916,6.690,149.253
C04767=1104.332,10.808,-53.027,179.916,6.686,149.252
C04768=1104.337,10.558,-53.011,179.915,6.681,149.252
C04769=1104.341,10.309,-52.996,179.915,6.676,149.251
C04770=1104.346,10.094,-52.983,179.914,6.673,149.250
C04771=1104.350,9.880,-52.970,179.914,6.669,149.249
C04772=1104.355,9.667,-52.957,179.914,6.665,149.248
C04773=1104.359,9.453,-52.945,179.914,6.661,149.248
C04774=1104.363,9.239,-52.932,179.913,6.657,149.247
C04775=1104.368,9.025,-52.919,179.913,6.653,149.246
C04776=1104.371,8.811,-52.906,179.913,6.650,149.245
C04777=1104.376,8.597,-52.893,179.912,6.646,149.245
C04778=1104.381,8.348,-52.878,179.912,6.641,149.244
C04779=1104.386,8.098,-52.864,179.911,6.637,149.243
C04780=1104.391,7.849,-52.848,179.911,6.632,149.242
C04781=1104.395,7.599,-52.833,179.910,6.628,149.241
C04782=1104.401,7.349,-52.818,179.909,6.623,149.240
C04783=1104.406,7.100,-52.803,179.908,6.618,149.240
C04784=1104.410,6.851,-52.788,179.908,6.613,149.239
C04785=1104.416,6.601,-52.773,179.907,6.609,149.238
C04786=1104.421,6.352,-52.758,179.906,6.604,149.237
C04787=1104.426,6.102,-52.744,179.906,6.600,149.236
C04788=1104.431,5.852,-52.728,179.905,6.595,149.235
C04789=1104.436,5.603,-52.714,179.904,6.590,149.235
C04790=1104.441,5.353,-52.698,179.903,6.585,149.234
C04791=1104.446,5.104,-52.684,179.903,6.580,149.233
C04792=1104.451,4.855,-52.669,179.902,6.576,149.232
C04793=1104.456,4.605,-52.654,179.901,6.571,149.231
C04794=1104.461,4.355,-52.639,179.900,6.567,149.230
C04795=1104.466,4.106,-52.624,179.901,6.563,149.230
C04796=1104.471,3.857,-52.610,179.900,6.558,149.229
C04797=1104.477,3.607,-52.595,179.899,6.554,149.228
C04798=1104.481,3.358,-52.580,179.898,6.549,149.227
C04799=1104.486,3.108,-52.566,179.898,6.544,149.226
C04800=1104.491,2.859,-52.551,179.897,6.540,149.226
C04801=1104.497,2.609,-52.536,179.896,6.535,149.225
C04802=1104.501,2.360,-52.521,179.896,6.531,149.224
C04803=1104.506,2.110,-52.506,179.895,6.526,149.223
C04804=1104.511,1.861,-52.491,179.894,6.522,149.222
C04805=1104.516,1.611,-52.477,179.894,6.517,149.221
C04806=1104.521,1.361,-52.462,179.893,6.512,149.220
C04807=1104.526,1.112,-52.447,179.892,6.508,149.220
C04808=1104.531,0.862,-52.433,179.892,6.503,149.219
C04809=1104.536,0.613,-52.419,179.891,6.498,149.218
C04810=1104.541,0.363,-52.403,179.891,6.494,149.217
C04811=1104.546,0.113,-52.389,179.890,6.489,149.216
C04812=1104.551,-0.136,-52.375,179.889,6.485,149.216
C04813=1104.556,-0.385,-52.360,179.889,6.480,149.215
C04814=1104.561,-0.635,-52.345,179.888,6.476,149.214
C04815=1104.567,-0.885,-52.330,179.887,6.471,149.213
C04816=1104.571,-1.134,-52.315,179.887,6.467,149.212
C04817=1104.576,-1.384,-52.301,179.886,6.463,149.212
C04818=1104.582,-1.633,-52.287,179.886,6.458,149.211
C04819=1104.587,-1.883,-52.273,179.885,6.453,149.210
C04820=1104.591,-2.132,-52.258,179.885,6.449,149.209
C04821=1104.596,-2.381,-52.244,179.884,6.444,149.208
C04822=1104.602,-2.631,-52.229,179.883,6.439,149.207
C04823=1104.607,-2.881,-52.215,179.883,6.435,149.206
C04824=1104.612,-3.130,-52.200,179.882,6.430,149.206
C04825=1104.617,-3.380,-52.185,179.881,6.426,149.205
C04826=1104.621,-3.594,-52.173,179.881,6.422,149.204
C04827=1104.625,-3.808,-52.161,179.881,6.418,149.203
C04828=1104.629,-4.022,-52.149,179.880,6.414,149.203
C04829=1104.634,-4.236,-52.136,179.879,6.410,149.202
C04830=1104.639,-4.450,-52.124,179.879,6.407,149.201
C04831=1104.643,-4.664,-52.111,179.878,6.403,149.201
C04832=1104.647,-4.879,-52.099,179.878,6.399,149.200
C04833=1104.652,-5.092,-52.087,179.878,6.395,149.199
C04834=1104.656,-5.342,-52.072,179.877,6.391,149.198
C04835=1104.661,-5.591,-52.058,179.876,6.386,149.197
C04836=1104.666,-5.841,-52.044,179.876,6.381,149.197
C04837=1104.672,-6.090,-52.030,179.875,6.377,149.196
C04838=1104.677,-6.340,-52.015,179.874,6.372,149.195
C04839=1104.682,-6.589,-52.001,179.874,6.368,149.194
C04840=1104.686,-6.839,-51.987,179.874,6.364,149.193
C04841=1104.691,-7.089,-51.972,179.873,6.359,149.192
C04842=1104.697,-7.338,-51.959,179.872,6.355,149.192
C04843=1104.702,-7.588,-51.944,179.872,6.350,149.191
C04844=1104.707,-7.837,-51.930,179.871,6.345,149.190
C04845=1104.712,-8.087,-51.916,179.871,6.340,149.189
C04846=1104.717,-8.337,-51.901,179.870,6.336,149.188
C04847=1104.722,-8.586,-51.888,179.870,6.332,149.187
C04848=1104.727,-8.835,-51.873,179.869,6.327,149.187
C04849=1104.732,-9.085,-51.859,179.869,6.323,149.186
C04850=1104.737,-9.335,-51.845,179.868,6.318,149.185
C04851=1104.742,-9.585,-51.830,179.867,6.314,149.184
C04852=1104.748,-9.834,-51.817,179.867,6.309,149.183
C04853=1104.752,-10.083,-51.803,179.866,6.304,149.182
C04854=1104.757,-10.333,-51.789,179.866,6.301,149.182
C04855=1104.762,-10.582,-51.774,179.865,6.296,149.181
C04856=1104.767,-10.831,-51.760,179.865,6.291,149.180
C04857=1104.772,-11.081,-51.746,179.864,6.287,149.179
C04858=1104.777,-11.331,-51.732,179.864,6.282,149.178
C04859=1104.782,-11.580,-51.718,179.863,6.278,149.177
C04860=1104.788,-11.829,-51.704,179.863,6.274,149.176
C04861=1104.793,-12.079,-51.689,179.862,6.269,149.176
C04862=1104.797,-12.329,-51.676,179.862,6.264,149.175
C04863=1104.802,-12.579,-51.662,179.861,6.259,149.174
C04864=1104.808,-12.828,-51.648,179.861,6.255,149.173
C04865=1104.813,-13.078,-51.634,179.860,6.250,149.172
C04866=1104.818,-13.327,-51.620,179.860,6.246,149.171
C04867=1104.823,-13.577,-51.605,179.860,6.242,149.170
C04868=1104.828,-13.826,-51.592,179.859,6.237,149.169
C04869=1104.833,-14.076,-51.578,179.859,6.232,149.169
C04870=1104.838,-14.326,-51.564,179.858,6.228,149.168
C04871=1104.843,-14.575,-51.550,179.858,6.223,149.167
C04872=1104.848,-14.825,-51.536,179.857,6.219,149.166
C04873=1104.852,-15.074,-51.522,179.857,6.215,149.165
C04874=1104.858,-15.324,-51.509,179.856,6.210,149.164
C04875=1104.863,-15.573,-51.495,179.856,6.205,149.163
C04876=1104.868,-15.823,-51.481,179.855,6.200,149.162
C04877=1104.874,-16.072,-51.467,179.855,6.196,149.162
C04878=1104.878,-16.322,-51.454,179.855,6.192,149.161
C04879=1104.883,-16.572,-51.439,179.854,6.187,149.160
C04880=1104.889,-16.821,-51.426,179.854,6.182,149.159
C04881=1104.894,-17.071,-51.412,179.853,6.178,149.158
C04882=1104.898,-17.285,-51.401,179.853,6.174,149.157
C04883=1104.902,-17.499,-51.389,179.853,6.171,149.157
C04884=1104.907,-17.713,-51.376,179.852,6.166,149.156
C04885=1104.911,-17.928,-51.365,179.852,6.162,149.155
C04886=1104.915,-18.142,-51.353,179.852,6.158,149.154
C04887=1104.920,-18.356,-51.341,179.852,6.155,149.153
C04888=1104.924,-18.569,-51.329,179.851,6.150,149.153
C04889=1104.928,-18.784,-51.318,179.851,6.147,149.152
C04890=1104.933,-19.034,-51.304,179.850,6.142,149.151
C04891=1104.939,-19.283,-51.291,179.850,6.137,149.150
C04892=1104.943,-19.533,-51.277,179.849,6.132,149.149
C04893=1104.949,-19.782,-51.263,179.849,6.128,149.148
C04894=1104.954,-20.032,-51.249,179.849,6.124,149.147
C04895=1104.958,-20.281,-51.236,179.848,6.119,149.146
C04896=1104.964,-20.531,-51.222,179.848,6.114,149.146
C04897=1104.969,-20.781,-51.208,179.847,6.110,149.145
C04898=1104.974,-21.029,-51.195,179.848,6.106,149.144
C04899=1104.979,-21.280,-51.181,179.847,6.101,149.143
C04900=1104.985,-21.529,-51.167,179.847,6.096,149.142
C04901=1104.989,-21.779,-51.154,179.846,6.091,149.141
C04902=1104.994,-22.028,-51.140,179.846,6.086,149.140
C04903=1104.999,-22.278,-51.128,179.846,6.082,149.139
C04904=1105.004,-22.527,-51.113,179.846,6.078,149.138
C04905=1105.010,-22.777,-51.100,179.845,6.073,149.137
C04906=1105.014,-23.026,-51.086,179.845,6.068,149.136
C04907=1105.020,-23.276,-51.073,179.844,6.064,149.135
C04908=1105.025,-23.525,-51.060,179.844,6.059,149.135
C04909=1105.030,-23.775,-51.046,179.844,6.054,149.133
C04910=1105.035,-24.025,-51.032,179.844,6.050,149.132
C04911=1105.040,-24.274,-51.019,179.844,6.045,149.132
C04912=1105.046,-24.524,-51.006,179.843,6.040,149.131
C04913=1105.051,-24.773,-50.993,179.843,6.036,149.130
C04914=1105.056,-25.023,-50.979,179.842,6.031,149.129
C04915=1105.061,-25.272,-50.966,179.842,6.026,149.128
C04916=1105.066,-25.523,-50.952,179.842,6.022,149.127
C04917=1105.071,-25.772,-50.940,179.842,6.017,149.126
C04918=1105.076,-26.022,-50.925,179.842,6.012,149.125
C04919=1105.081,-26.271,-50.913,179.841,6.007,149.124
C04920=1105.086,-26.521,-50.898,179.841,6.003,149.123
C04921=1105.091,-26.770,-50.886,179.841,5.999,149.122
C04922=1105.096,-27.020,-50.872,179.840,5.994,149.121
C04923=1105.101,-27.269,-50.859,179.841,5.989,149.120
C04924=1105.107,-27.519,-50.845,179.841,5.985,149.119
C04925=1105.112,-27.769,-50.833,179.840,5.980,149.118
C04926=1105.117,-28.018,-50.818,179.840,5.975,149.117
C04927=1105.122,-28.268,-50.806,179.840,5.971,149.116
C04928=1105.127,-28.518,-50.792,179.839,5.967,149.116
C04929=1105.132,-28.767,-50.779,179.839,5.962,149.115
C04930=1105.137,-29.017,-50.765,179.839,5.958,149.114
C04931=1105.142,-29.266,-50.753,179.839,5.953,149.113
C04932=1105.147,-29.517,-50.739,179.838,5.949,149.112
C04933=1105.152,-29.765,-50.726,179.838,5.945,149.111
C04934=1105.157,-30.015,-50.713,179.838,5.940,149.110
C04935=1105.163,-30.265,-50.700,179.837,5.935,149.109
C04936=1105.168,-30.514,-50.687,179.837,5.931,149.108
C04937=1105.173,-30.764,-50.673,179.837,5.927,149.107
C04938=1105.177,-30.978,-50.662,179.837,5.923,149.106
C04939=1105.182,-31.193,-50.651,179.837,5.919,149.106
C04940=1105.185,-31.406,-50.639,179.836,5.915,149.105
C04941=1105.190,-31.621,-50.628,179.836,5.911,149.104
C04942=1105.194,-31.835,-50.617,179.836,5.907,149.103
C04943=1105.199,-32.050,-50.606,179.835,5.904,149.103
C04944=1105.203,-32.264,-50.594,179.835,5.900,149.102
C04945=1105.207,-32.478,-50.583,179.835,5.896,149.101
C04946=1105.212,-32.727,-50.571,179.835,5.891,149.100
C04947=1105.218,-32.977,-50.558,179.834,5.887,149.099
C04948=1105.223,-33.227,-50.545,179.834,5.883,149.098
C04949=1105.228,-33.476,-50.531,179.834,5.878,149.098
C04950=1105.234,-33.725,-50.518,179.833,5.873,149.097
C04951=1105.238,-33.975,-50.505,179.833,5.870,149.096
C04952=1105.244,-34.225,-50.492,179.833,5.865,149.095
C04953=1105.248,-34.475,-50.479,179.832,5.860,149.094
C04954=1105.254,-34.724,-50.466,179.832,5.856,149.093
C04955=1105.259,-34.973,-50.454,179.832,5.852,149.092
C04956=1105.264,-35.224,-50.440,179.831,5.847,149.091
C04957=1105.269,-35.473,-50.428,179.831,5.842,149.091
C04958=1105.274,-35.722,-50.415,179.831,5.838,149.090
C04959=1105.279,-35.973,-50.401,179.831,5.833,149.089
C04960=1105.285,-36.222,-50.389,179.830,5.829,149.088
C04961=1105.290,-36.471,-50.376,179.830,5.824,149.087
C04962=1105.294,-36.721,-50.363,179.830,5.820,149.086
C04963=1105.300,-36.971,-50.350,179.829,5.816,149.085
C04964=1105.305,-37.220,-50.337,179.829,5.811,149.084
C04965=1105.310,-37.470,-50.324,179.828,5.806,149.083
C04966=1105.315,-37.720,-50.312,179.828,5.802,149.083
C04967=1105.321,-37.969,-50.299,179.828,5.798,149.082
C04968=1105.326,-38.219,-50.286,179.828,5.792,149.080
C04969=1105.330,-38.469,-50.273,179.827,5.788,149.080
C04970=1105.335,-38.718,-50.261,179.827,5.783,149.079
C04971=1105.341,-38.968,-50.247,179.827,5.778,149.078
C04972=1105.346,-39.218,-50.234,179.827,5.774,149.077
C04973=1105.351,-39.467,-50.222,179.826,5.770,149.076
C04974=1105.356,-39.716,-50.209,179.826,5.765,149.075
C04975=1105.361,-39.966,-50.197,179.825,5.760,149.074
C04976=1105.366,-40.216,-50.183,179.825,5.755,149.073
C04977=1105.372,-40.465,-50.170,179.825,5.750,149.072
C04978=1105.377,-40.715,-50.158,179.825,5.746,149.071
C04979=1105.382,-40.964,-50.146,179.824,5.741,149.070
C04980=1105.387,-41.214,-50.133,179.824,5.736,149.069
C04981=1105.392,-41.464,-50.120,179.824,5.731,149.068
C04982=1105.398,-41.713,-50.107,179.823,5.726,149.067
C04983=1105.403,-41.963,-50.095,179.823,5.721,149.066
C04984=1105.407,-42.213,-50.082,179.823,5.716,149.065
C04985=1105.413,-42.463,-50.070,179.822,5.712,149.064
C04986=1105.418,-42.712,-50.057,179.823,5.706,149.063
C04987=1105.423,-42.961,-50.044,179.823,5.703,149.062
C04988=1105.428,-43.211,-50.032,179.823,5.697,149.061
C04989=1105.433,-43.461,-50.019,179.823,5.693,149.060
C04990=1105.438,-43.711,-50.007,179.823,5.688,149.059
C04991=1105.444,-43.960,-49.994,179.823,5.683,149.058
C04992=1105.449,-44.210,-49.981,179.824,5.679,149.057
C04993=1105.454,-44.460,-49.968,179.824,5.674,149.056
C04994=1105.458,-44.673,-49.958,179.824,5.670,149.055
C04995=1105.463,-44.888,-49.948,179.824,5.666,149.054
C04996=1105.467,-45.103,-49.937,179.824,5.662,149.053
C04997=1105.471,-45.317,-49.926,179.824,5.658,149.052
C04998=1105.475,-45.531,-49.915,179.824,5.653,149.051
C04999=1105.480,-45.745,-49.905,179.824,5.649,149.050
C05000=1105.485,-45.959,-49.893,179.824,5.645,149.049
C05001=1105.489,-46.173,-49.883,179.825,5.642,149.048
C05002=1105.494,-46.423,-49.871,179.825,5.636,149.047
C05003=1105.499,-46.673,-49.858,179.825,5.632,149.046
C05004=1105.504,-46.923,-49.845,179.825,5.627,149.045
C05005=1105.509,-47.173,-49.833,179.825,5.623,149.044
C05006=1105.514,-47.422,-49.821,179.826,5.618,149.043
C05007=1105.520,-47.671,-49.808,179.825,5.613,149.042
C05008=1105.525,-47.921,-49.796,179.826,5.609,149.041
C05009=1105.530,-48.170,-49.784,179.826,5.604,149.039
C05010=1105.535,-48.420,-49.771,179.826,5.599,149.038
C05011=1105.540,-48.670,-49.759,179.826,5.595,149.037
C05012=1105.545,-48.920,-49.746,179.826,5.589,149.036
C05013=1105.551,-49.170,-49.734,179.826,5.584,149.035
C05014=1105.556,-49.419,-49.722,179.826,5.580,149.034
C05015=1105.561,-49.668,-49.709,179.827,5.575,149.033
C05016=1105.566,-49.918,-49.697,179.827,5.571,149.032
C05017=1105.571,-50.168,-49.685,179.827,5.566,149.031
C05018=1105.577,-50.417,-49.673,179.827,5.561,149.030
C05019=1105.581,-50.667,-49.660,179.828,5.557,149.029
C05020=1105.587,-50.917,-49.648,179.827,5.552,149.028
C05021=1105.592,-51.167,-49.635,179.827,5.547,149.027
C05022=1105.597,-51.416,-49.623,179.828,5.543,149.025
C05023=1105.602,-51.666,-49.611,179.827,5.538,149.024
C05024=1105.607,-51.915,-49.599,179.828,5.533,149.023
C05025=1105.612,-52.165,-49.587,179.828,5.528,149.022
C05026=1105.617,-52.414,-49.574,179.828,5.524,149.021
C05027=1105.623,-52.664,-49.563,179.828,5.519,149.020
C05028=1105.628,-52.914,-49.550,179.829,5.514,149.019
C05029=1105.633,-53.163,-49.538,179.828,5.509,149.018
C05030=1105.638,-53.413,-49.525,179.828,5.504,149.017
C05031=1105.643,-53.663,-49.513,179.829,5.500,149.016
C05032=1105.648,-53.913,-49.501,179.828,5.495,149.015
C05033=1105.653,-54.162,-49.489,179.829,5.491,149.014
C05034=1105.659,-54.412,-49.477,179.829,5.486,149.012
C05035=1105.664,-54.662,-49.465,179.829,5.481,149.012
C05036=1105.669,-54.912,-49.453,179.830,5.477,149.010
C05037=1105.674,-55.161,-49.440,179.830,5.472,149.009
C05038=1105.680,-55.411,-49.428,179.829,5.467,149.008
C05039=1105.684,-55.660,-49.416,179.830,5.463,149.007
C05040=1105.690,-55.910,-49.405,179.830,5.458,149.006
C05041=1105.695,-56.160,-49.393,179.830,5.453,149.005
C05042=1105.700,-56.409,-49.380,179.830,5.448,149.004
C05043=1105.706,-56.659,-49.368,179.830,5.444,149.003
C05044=1105.710,-56.908,-49.356,179.830,5.438,149.002
C05045=1105.715,-57.158,-49.344,179.831,5.434,149.001
C05046=1105.721,-57.408,-49.332,179.830,5.429,149.000
C05047=1105.726,-57.657,-49.320,179.830,5.424,148.999
C05048=1105.731,-57.907,-49.308,179.831,5.420,148.998
C05049=1105.736,-58.157,-49.297,179.831,5.415,148.997
C05050=1105.740,-58.371,-49.286,179.831,5.411,148.996
C05051=1105.744,-58.586,-49.276,179.831,5.407,148.995
C05052=1105.750,-58.800,-49.265,179.831,5.403,148.994
C05053=1105.754,-59.014,-49.255,179.831,5.399,148.993
C05054=1105.758,-59.229,-49.244,179.831,5.395,148.992
C05055=1105.763,-59.443,-49.235,179.831,5.391,148.991
C05056=1105.767,-59.657,-49.224,179.831,5.387,148.990
C05057=1105.771,-59.872,-49.214,179.831,5.383,148.989
C05058=1105.776,-60.122,-49.203,179.831,5.378,148.988
C05059=1105.781,-60.371,-49.190,179.831,5.373,148.987
C05060=1105.787,-60.621,-49.178,179.830,5.369,148.986
C05061=1105.792,-60.871,-49.166,179.831,5.363,148.985
C05062=1105.797,-61.120,-49.155,179.830,5.359,148.984
C05063=1105.802,-61.370,-49.143,179.829,5.353,148.983
C05064=1105.807,-61.620,-49.130,179.829,5.348,148.982
C05065=1105.813,-61.869,-49.119,179.829,5.343,148.981
C05066=1105.818,-62.119,-49.108,179.829,5.338,148.980
C05067=1105.823,-62.368,-49.096,179.829,5.333,148.979
C05068=1105.828,-62.618,-49.084,179.829,5.328,148.978
C05069=1105.833,-62.867,-49.072,179.828,5.324,148.977
C05070=1105.839,-63.117,-49.060,179.829,5.318,148.976
C05071=1105.843,-63.367,-49.049,179.828,5.314,148.975
C05072=1105.849,-63.617,-49.037,179.828,5.309,148.974
C05073=1105.854,-63.867,-49.025,179.828,5.304,148.973
C05074=1105.859,-64.116,-49.014,179.828,5.299,148.972
C05075=1105.864,-64.366,-49.002,179.828,5.294,148.971
C05076=1105.869,-64.615,-48.990,179.828,5.289,148.970
C05077=1105.875,-64.865,-48.978,179.827,5.284,148.969
C05078=1105.880,-65.115,-48.966,179.827,5.279,148.968
C05079=1105.885,-65.364,-48.955,179.828,5.274,148.966
C05080=1105.890,-65.614,-48.943,179.827,5.269,148.965
C05081=1105.895,-65.864,-48.932,179.827,5.264,148.964
C05082=1105.900,-66.114,-48.920,179.827,5.258,148.963
C05083=1105.906,-66.364,-48.908,179.826,5.253,148.962
C05084=1105.911,-66.613,-48.897,179.827,5.248,148.961
C05085=1105.917,-66.863,-48.885,179.827,5.243,148.960
C05086=1105.921,-67.112,-48.874,179.826,5.238,148.959
C05087=1105.927,-67.362,-48.862,179.826,5.233,148.958
C05088=1105.931,-67.612,-48.851,179.827,5.228,148.957
C05089=1105.937,-67.862,-48.839,179.826,5.223,148.956
C05090=1105.942,-68.111,-48.828,179.826,5.218,148.954
C05091=1105.948,-68.360,-48.816,179.826,5.213,148.953
C05092=1105.952,-68.610,-48.805,179.827,5.208,148.952
C05093=1105.958,-68.860,-48.793,179.826,5.203,148.951
C05094=1105.962,-69.110,-48.782,179.826,5.198,148.950
C05095=1105.968,-69.360,-48.770,179.826,5.193,148.949
C05096=1105.973,-69.609,-48.759,179.827,5.188,148.948
C05097=1105.979,-69.858,-48.747,179.827,5.182,148.947
C05098=1105.983,-70.108,-48.736,179.826,5.178,148.946
C05099=1105.989,-70.358,-48.724,179.826,5.173,148.944
C05100=1105.993,-70.608,-48.712,179.827,5.167,148.943
C05101=1106.000,-70.858,-48.702,179.827,5.162,148.942
C05102=1106.004,-71.107,-48.690,179.827,5.157,148.941
C05103=1106.010,-71.357,-48.678,179.827,5.152,148.940
C05104=1106.015,-71.607,-48.667,179.827,5.147,148.939
C05105=1106.020,-71.856,-48.656,179.827,5.142,148.938
C05106=1106.024,-72.070,-48.646,179.827,5.137,148.936
C05107=1106.028,-72.285,-48.636,179.827,5.133,148.936
C05108=1106.033,-72.500,-48.627,179.827,5.128,148.935
C05109=1106.038,-72.714,-48.617,179.827,5.124,148.934
C05110=1106.043,-72.929,-48.607,179.827,5.120,148.933
C05111=1106.046,-73.143,-48.598,179.827,5.115,148.932
C05112=1106.051,-73.357,-48.588,179.827,5.110,148.931
C05113=1106.056,-73.572,-48.578,179.827,5.107,148.930
C05114=1106.061,-73.821,-48.567,179.827,5.101,148.929
C05115=1106.067,-74.072,-48.556,179.828,5.096,148.927
C05116=1106.071,-74.321,-48.545,179.828,5.091,148.926
C05117=1106.076,-74.571,-48.533,179.828,5.086,148.925
C05118=1106.082,-74.820,-48.522,179.828,5.081,148.924
C05119=1106.087,-75.070,-48.511,179.828,5.076,148.923
C05120=1106.092,-75.320,-48.499,179.828,5.071,148.922
C05121=1106.098,-75.569,-48.488,179.828,5.065,148.920
C05122=1106.102,-75.819,-48.477,179.829,5.060,148.919
C05123=1106.108,-76.069,-48.466,179.829,5.055,148.918
C05124=1106.113,-76.318,-48.455,179.829,5.050,148.917
C05125=1106.118,-76.568,-48.444,179.829,5.045,148.916
C05126=1106.124,-76.818,-48.432,179.829,5.040,148.914
C05127=1106.129,-77.067,-48.422,179.829,5.035,148.913
C05128=1106.134,-77.317,-48.410,179.829,5.029,148.912
C05129=1106.139,-77.567,-48.400,179.830,5.024,148.911
C05130=1106.145,-77.816,-48.388,179.830,5.019,148.910
C05131=1106.150,-78.066,-48.377,179.830,5.014,148.909
C05132=1106.155,-78.316,-48.366,179.830,5.009,148.907
C05133=1106.161,-78.566,-48.355,179.830,5.004,148.906
C05134=1106.165,-78.815,-48.344,179.830,4.999,148.905
C05135=1106.170,-79.065,-48.333,179.831,4.993,148.904
C05136=1106.176,-79.314,-48.322,179.831,4.988,148.903
C05137=1106.181,-79.565,-48.311,179.831,4.983,148.902
C05138=1106.186,-79.815,-48.300,179.831,4.978,148.900
C05139=1106.191,-80.063,-48.289,179.831,4.973,148.899
C05140=1106.196,-80.314,-48.278,179.831,4.968,148.898
C05141=1106.202,-80.563,-48.267,179.832,4.962,148.897
C05142=1106.207,-80.813,-48.256,179.833,4.958,148.895
C05143=1106.212,-81.063,-48.245,179.833,4.953,148.894
C05144=1106.218,-81.312,-48.234,179.833,4.948,148.893
C05145=1106.223,-81.562,-48.223,179.833,4.942,148.892
C05146=1106.228,-81.813,-48.212,179.833,4.937,148.891
C05147=1106.233,-82.061,-48.201,179.834,4.932,148.890
C05148=1106.238,-82.312,-48.191,179.834,4.927,148.888
C05149=1106.244,-82.561,-48.180,179.834,4.922,148.887
C05150=1106.249,-82.811,-48.169,179.834,4.917,148.886
C05151=1106.255,-83.060,-48.157,179.835,4.911,148.885
C05152=1106.260,-83.310,-48.147,179.835,4.906,148.883
C05153=1106.264,-83.560,-48.136,179.836,4.902,148.882
C05154=1106.270,-83.810,-48.125,179.836,4.897,148.881
C05155=1106.275,-84.059,-48.114,179.836,4.891,148.880
C05156=1106.280,-84.309,-48.104,179.836,4.886,148.879
C05157=1106.286,-84.559,-48.092,179.836,4.881,148.877
C05158=1106.291,-84.808,-48.082,179.837,4.876,148.876
C05159=1106.296,-85.058,-48.071,179.837,4.871,148.875
C05160=1106.301,-85.308,-48.060,179.838,4.867,148.874
C05161=1106.307,-85.558,-48.050,179.838,4.861,148.873
C05162=1106.311,-85.772,-48.040,179.838,4.856,148.872
C05163=1106.315,-85.987,-48.031,179.838,4.852,148.871
C05164=1106.320,-86.201,-48.022,179.839,4.848,148.869
C05165=1106.324,-86.416,-48.012,179.839,4.843,148.868
C05166=1106.329,-86.630,-48.003,179.839,4.839,148.867
C05167=1106.333,-86.845,-47.994,179.840,4.835,148.866
C05168=1106.338,-87.060,-47.985,179.840,4.831,148.865
C05169=1106.342,-87.274,-47.976,179.840,4.826,148.864
C05170=1106.347,-87.524,-47.965,179.841,4.821,148.863
C05171=1106.353,-87.773,-47.955,179.841,4.816,148.862
C05172=1106.358,-88.023,-47.944,179.841,4.811,148.861
C05173=1106.363,-88.273,-47.934,179.841,4.806,148.859
C05174=1106.369,-88.523,-47.922,179.842,4.801,148.858
C05175=1106.374,-88.772,-47.912,179.842,4.797,148.857
C05176=1106.379,-89.022,-47.901,179.843,4.791,148.856
C05177=1106.384,-89.271,-47.890,179.843,4.786,148.854
C05178=1106.389,-89.521,-47.880,179.843,4.781,148.853
C05179=1106.395,-89.771,-47.869,179.844,4.776,148.852
C05180=1106.400,-90.021,-47.859,179.844,4.771,148.851
C05181=1106.405,-90.270,-47.848,179.845,4.766,148.850
C05182=1106.410,-90.520,-47.837,179.845,4.761,148.849
C05183=1106.416,-90.770,-47.827,179.846,4.757,148.847
C05184=1106.421,-91.020,-47.817,179.846,4.752,148.846
C05185=1106.426,-91.269,-47.806,179.846,4.746,148.845
C05186=1106.431,-91.519,-47.795,179.846,4.741,148.844
C05187=1106.437,-91.769,-47.785,179.847,4.737,148.843
C05188=1106.442,-92.019,-47.774,179.847,4.732,148.841
C05189=1106.447,-92.269,-47.764,179.848,4.726,148.840
C05190=1106.452,-92.517,-47.754,179.849,4.722,148.839
C05191=1106.457,-92.768,-47.743,179.849,4.717,148.838
C05192=1106.463,-93.017,-47.733,179.849,4.712,148.836
C05193=1106.468,-93.267,-47.722,179.850,4.707,148.835
C05194=1106.473,-93.517,-47.712,179.850,4.702,148.834
C05195=1106.478,-93.767,-47.702,179.850,4.697,148.833
C05196=1106.483,-94.016,-47.691,179.851,4.693,148.832
C05197=1106.488,-94.266,-47.680,179.851,4.687,148.830
C05198=1106.494,-94.516,-47.670,179.851,4.682,148.829
C05199=1106.500,-94.765,-47.660,179.852,4.678,148.828
C05200=1106.505,-95.016,-47.649,179.852,4.673,148.827
C05201=1106.510,-95.265,-47.639,179.853,4.668,148.826
C05202=1106.515,-95.515,-47.628,179.853,4.663,148.825
C05203=1106.521,-95.765,-47.618,179.854,4.658,148.823
C05204=1106.525,-96.014,-47.608,179.854,4.653,148.822
C05205=1106.530,-96.264,-47.597,179.855,4.649,148.821
C05206=1106.536,-96.513,-47.587,179.855,4.644,148.820
C05207=1106.541,-96.764,-47.576,179.855,4.638,148.819
C05208=1106.547,-97.013,-47.566,179.855,4.633,148.817
C05209=1106.552,-97.263,-47.556,179.856,4.629,148.816
C05210=1106.557,-97.513,-47.545,179.856,4.624,148.815
C05211=1106.563,-97.762,-47.535,179.856,4.619,148.814
C05212=1106.568,-98.012,-47.526,179.857,4.614,148.813
C05213=1106.573,-98.262,-47.515,179.857,4.609,148.811
C05214=1106.578,-98.512,-47.505,179.858,4.604,148.810
C05215=1106.584,-98.761,-47.495,179.858,4.599,148.809
C05216=1106.589,-99.011,-47.484,179.859,4.594,148.808
C05217=1106.594,-99.261,-47.474,179.859,4.589,148.807
C05218=1106.599,-99.475,-47.466,179.859,4.585,148.806
C05219=1106.603,-99.690,-47.457,179.860,4.581,148.804
C05220=1106.608,-99.905,-47.447,179.860,4.576,148.803
C05221=1106.612,-100.119,-47.439,179.860,4.572,148.803
C05222=1106.617,-100.334,-47.431,179.860,4.568,148.802
C05223=1106.621,-100.549,-47.422,179.861,4.564,148.800
C05224=1106.626,-100.763,-47.412,179.861,4.560,148.799
C05225=1106.630,-100.977,-47.404,179.861,4.555,148.798
C05226=1106.636,-101.227,-47.394,179.862,4.551,148.797
C05227=1106.641,-101.477,-47.383,179.862,4.546,148.796
C05228=1106.646,-101.727,-47.374,179.862,4.541,148.795
C05229=1106.652,-101.977,-47.364,179.864,4.536,148.793
C05230=1106.657,-102.227,-47.353,179.864,4.531,148.792
C05231=1106.662,-102.476,-47.343,179.864,4.526,148.791
C05232=1106.667,-102.726,-47.334,179.864,4.520,148.790
C05233=1106.672,-102.976,-47.323,179.865,4.516,148.789
C05234=1106.678,-103.225,-47.313,179.865,4.511,148.787
C05235=1106.683,-103.475,-47.303,179.866,4.506,148.786
C05236=1106.687,-103.725,-47.293,179.866,4.501,148.785
C05237=1106.693,-103.975,-47.283,179.867,4.496,148.784
C05238=1106.699,-104.225,-47.273,179.867,4.491,148.783
C05239=1106.704,-104.474,-47.263,179.867,4.486,148.781
C05240=1106.709,-104.724,-47.253,179.867,4.481,148.780
C05241=1106.714,-104.974,-47.242,179.868,4.477,148.779
C05242=1106.720,-105.223,-47.232,179.868,4.471,148.778
C05243=1106.725,-105.474,-47.223,179.869,4.466,148.777
C05244=1106.730,-105.723,-47.213,179.869,4.461,148.775
C05245=1106.736,-105.973,-47.203,179.870,4.457,148.774
C05246=1106.741,-106.222,-47.193,179.870,4.452,148.773
C05247=1106.746,-106.472,-47.182,179.871,4.446,148.772
C05248=1106.751,-106.722,-47.173,179.871,4.441,148.770
C05249=1106.756,-106.972,-47.163,179.871,4.436,148.769
C05250=1106.762,-107.221,-47.153,179.872,4.431,148.768
C05251=1106.766,-107.471,-47.143,179.872,4.426,148.767
C05252=1106.772,-107.721,-47.134,179.873,4.421,148.766
C05253=1106.778,-107.971,-47.123,179.873,4.416,148.764
C05254=1106.783,-108.220,-47.114,179.874,4.412,148.763
C05255=1106.788,-108.470,-47.104,179.874,4.406,148.762
C05256=1106.793,-108.720,-47.094,179.874,4.401,148.761
C05257=1106.798,-108.970,-47.084,179.875,4.396,148.759
C05258=1106.804,-109.219,-47.074,179.875,4.391,148.758
C05259=1106.809,-109.468,-47.064,179.876,4.386,148.757
C05260=1106.815,-109.719,-47.055,179.876,4.381,148.756
C05261=1106.820,-109.969,-47.044,179.876,4.376,148.754
C05262=1106.825,-110.218,-47.035,179.877,4.371,148.753
C05263=1106.830,-110.468,-47.025,179.877,4.366,148.752
C05264=1106.835,-110.717,-47.016,179.877,4.361,148.751
C05265=1106.841,-110.967,-47.005,179.879,4.356,148.749
C05266=1106.845,-111.218,-46.996,179.879,4.351,148.748
C05267=1106.851,-111.467,-46.986,179.879,4.345,148.747
C05268=1106.857,-111.717,-46.976,179.879,4.340,148.746
C05269=1106.862,-111.967,-46.967,179.880,4.335,148.745
C05270=1106.867,-112.216,-46.957,179.880,4.331,148.743
C05271=1106.873,-112.466,-46.948,179.881,4.326,148.742
C05272=1106.878,-112.716,-46.937,179.881,4.320,148.741
C05273=1106.883,-112.966,-46.928,179.882,4.315,148.739
C05274=1106.887,-113.180,-46.920,179.882,4.311,148.739
C05275=1106.892,-113.395,-46.911,179.882,4.306,148.737
C05276=1106.897,-113.610,-46.903,179.883,4.302,148.736
C05277=1106.902,-113.824,-46.894,179.883,4.298,148.735
C05278=1106.906,-114.039,-46.886,179.884,4.294,148.734
C05279=1106.911,-114.254,-46.878,179.884,4.288,148.733
C05280=1106.915,-114.469,-46.870,179.884,4.284,148.732
C05281=1106.919,-114.683,-46.861,179.885,4.280,148.731
C05282=1106.924,-114.933,-46.852,179.885,4.275,148.730
C05283=1106.930,-115.183,-46.842,179.886,4.270,148.728
C05284=1106.935,-115.432,-46.833,179.886,4.265,148.727
C05285=1106.941,-115.682,-46.823,179.886,4.260,148.726
C05286=1106.946,-115.931,-46.813,179.887,4.254,148.724
C05287=1106.952,-116.182,-46.804,179.887,4.249,148.723
C05288=1106.956,-116.431,-46.794,179.888,4.244,148.722
C05289=1106.962,-116.682,-46.784,179.888,4.239,148.721
C05290=1106.967,-116.932,-46.776,179.889,4.234,148.719
C05291=1106.973,-117.181,-46.765,179.889,4.229,148.718
C05292=1106.978,-117.431,-46.756,179.890,4.223,148.717
C05293=1106.983,-117.680,-46.747,179.890,4.218,148.716
C05294=1106.988,-117.930,-46.737,179.891,4.213,148.714
C05295=1106.993,-118.180,-46.728,179.891,4.208,148.713
C05296=1106.999,-118.430,-46.718,179.891,4.202,148.712
C05297=1107.004,-118.679,-46.709,179.892,4.197,148.711
C05298=1107.010,-118.929,-46.699,179.892,4.192,148.709
C05299=1107.015,-119.179,-46.690,179.893,4.187,148.708
C05300=1107.020,-119.428,-46.681,179.894,4.182,148.707
C05301=1107.026,-119.678,-46.671,179.894,4.177,148.705
C05302=1107.031,-119.928,-46.662,179.895,4.172,148.704
C05303=1107.036,-120.177,-46.653,179.895,4.166,148.703
C05304=1107.041,-120.428,-46.643,179.896,4.161,148.701
C05305=1107.046,-120.678,-46.633,179.896,4.156,148.700
C05306=1107.051,-120.927,-46.624,179.896,4.151,148.699
C05307=1107.057,-121.178,-46.615,179.897,4.145,148.697
C05308=1107.062,-121.427,-46.605,179.897,4.140,148.696
C05309=1107.068,-121.677,-46.596,179.898,4.135,148.695
C05310=1107.073,-121.927,-46.587,179.899,4.129,148.694
C05311=1107.078,-122.176,-46.577,179.899,4.124,148.692
C05312=1107.083,-122.426,-46.568,179.899,4.119,148.691
C05313=1107.089,-122.676,-46.559,179.900,4.113,148.690
C05314=1107.094,-122.926,-46.550,179.900,4.108,148.688
C05315=1107.099,-123.175,-46.540,179.901,4.103,148.687
C05316=1107.105,-123.425,-46.531,179.901,4.097,148.686
C05317=1107.110,-123.675,-46.522,179.902,4.092,148.685
C05318=1107.115,-123.924,-46.512,179.902,4.087,148.683
C05319=1107.121,-124.175,-46.503,179.903,4.082,148.682
C05320=1107.126,-124.424,-46.494,179.903,4.076,148.680
C05321=1107.131,-124.674,-46.485,179.904,4.071,148.679
C05322=1107.136,-124.924,-46.476,179.905,4.065,148.678
C05323=1107.142,-125.174,-46.466,179.905,4.060,148.677
C05324=1107.147,-125.423,-46.457,179.905,4.055,148.675
C05325=1107.152,-125.673,-46.448,179.906,4.049,148.674
C05326=1107.158,-125.922,-46.440,179.906,4.044,148.673
C05327=1107.164,-126.173,-46.430,179.907,4.039,148.671
C05328=1107.169,-126.422,-46.420,179.907,4.034,148.670
C05329=1107.174,-126.672,-46.412,179.908,4.028,148.668
C05330=1107.179,-126.887,-46.404,179.909,4.024,148.667
C05331=1107.183,-127.101,-46.396,179.909,4.019,148.666
C05332=1107.188,-127.316,-46.388,179.910,4.015,148.665
C05333=1107.192,-127.531,-46.380,179.910,4.009,148.664
C05334=1107.197,-127.746,-46.373,179.910,4.005,148.663
C05335=1107.202,-127.961,-46.365,179.911,4.000,148.662
C05336=1107.206,-128.175,-46.357,179.912,3.996,148.660
C05337=1107.211,-128.390,-46.349,179.912,3.991,148.659
C05338=1106.788,-128.380,-46.375,179.919,3.995,148.658
C05339=1106.783,-128.166,-46.383,179.919,4.001,148.659
C05340=1106.779,-127.951,-46.391,179.918,4.005,148.660
C05341=1106.773,-127.737,-46.399,179.918,4.010,148.661
C05342=1106.769,-127.522,-46.406,179.917,4.014,148.663
C05343=1106.764,-127.307,-46.414,179.917,4.019,148.664
C05344=1106.760,-127.093,-46.422,179.917,4.023,148.665
C05345=1106.755,-126.878,-46.429,179.916,4.028,148.666
C05346=1106.751,-126.663,-46.437,179.915,4.033,148.667
C05347=1106.746,-126.413,-46.446,179.915,4.038,148.668
C05348=1106.740,-126.163,-46.456,179.914,4.043,148.670
C05349=1106.735,-125.913,-46.465,179.914,4.049,148.671
C05350=1106.730,-125.664,-46.474,179.913,4.054,148.673
C05351=1106.724,-125.414,-46.483,179.913,4.059,148.674
C05352=1106.719,-125.164,-46.493,179.912,4.065,148.675
C05353=1106.713,-124.914,-46.502,179.912,4.070,148.676
C05354=1106.709,-124.665,-46.511,179.911,4.076,148.678
C05355=1106.703,-124.415,-46.521,179.911,4.081,148.679
C05356=1106.697,-124.165,-46.530,179.910,4.086,148.680
C05357=1106.692,-123.915,-46.539,179.910,4.091,148.682
C05358=1106.687,-123.666,-46.548,179.909,4.097,148.683
C05359=1106.682,-123.416,-46.558,179.908,4.102,148.685
C05360=1106.676,-123.166,-46.567,179.908,4.107,148.686
C05361=1106.672,-122.917,-46.576,179.908,4.112,148.687
C05362=1106.666,-122.666,-46.586,179.907,4.118,148.688
C05363=1106.660,-122.417,-46.595,179.907,4.123,148.690
C05364=1106.656,-122.167,-46.604,179.906,4.129,148.691
C05365=1106.650,-121.917,-46.614,179.906,4.134,148.692
C05366=1106.645,-121.667,-46.623,179.905,4.139,148.694
C05367=1106.640,-121.418,-46.632,179.905,4.145,148.695
C05368=1106.634,-121.168,-46.642,179.904,4.150,148.696
C05369=1106.629,-120.917,-46.651,179.903,4.154,148.697
C05370=1106.624,-120.668,-46.661,179.903,4.160,148.699
C05371=1106.618,-120.418,-46.670,179.902,4.165,148.700
C05372=1106.614,-120.169,-46.680,179.902,4.170,148.701
C05373=1106.608,-119.919,-46.689,179.901,4.175,148.703
C05374=1106.602,-119.669,-46.698,179.901,4.181,148.704
C05375=1106.598,-119.420,-46.708,179.901,4.186,148.705
C05376=1106.592,-119.169,-46.717,179.900,4.191,148.707
C05377=1106.587,-118.920,-46.727,179.900,4.196,148.708
C05378=1106.581,-118.670,-46.736,179.899,4.202,148.709
C05379=1106.576,-118.420,-46.745,179.899,4.207,148.711
C05380=1106.571,-118.171,-46.755,179.898,4.212,148.712
C05381=1106.565,-117.921,-46.764,179.897,4.217,148.713
C05382=1106.560,-117.672,-46.774,179.897,4.222,148.714
C05383=1106.555,-117.421,-46.784,179.896,4.227,148.716
C05384=1106.550,-117.171,-46.793,179.896,4.232,148.717
C05385=1106.544,-116.921,-46.803,179.896,4.238,148.718
C05386=1106.539,-116.672,-46.812,179.895,4.243,148.720
C05387=1106.533,-116.422,-46.822,179.895,4.248,148.721
C05388=1106.528,-116.173,-46.832,179.895,4.253,148.722
C05389=1106.523,-115.922,-46.841,179.894,4.259,148.723
C05390=1106.518,-115.673,-46.851,179.893,4.263,148.724
C05391=1106.512,-115.423,-46.860,179.893,4.268,148.726
C05392=1106.507,-115.174,-46.870,179.892,4.274,148.727
C05393=1106.502,-114.923,-46.880,179.892,4.279,148.728
C05394=1106.497,-114.674,-46.889,179.892,4.284,148.730
C05395=1106.492,-114.459,-46.898,179.891,4.288,148.731
C05396=1106.488,-114.245,-46.906,179.891,4.292,148.732
C05397=1106.483,-114.030,-46.914,179.890,4.297,148.733
C05398=1106.478,-113.815,-46.922,179.890,4.301,148.734
C05399=1106.473,-113.600,-46.931,179.889,4.306,148.735
C05400=1106.469,-113.386,-46.939,179.889,4.311,148.736
C05401=1106.465,-113.171,-46.948,179.889,4.315,148.737
C05402=1106.460,-112.956,-46.956,179.888,4.319,148.738
C05403=1106.455,-112.707,-46.965,179.888,4.324,148.739
C05404=1106.450,-112.457,-46.975,179.888,4.329,148.741
C05405=1106.445,-112.208,-46.985,179.887,4.335,148.742
C05406=1106.439,-111.958,-46.994,179.887,4.340,148.743
C05407=1106.434,-111.707,-47.005,179.886,4.344,148.745
C05408=1106.429,-111.458,-47.015,179.886,4.349,148.746
C05409=1106.423,-111.208,-47.024,179.885,4.354,148.747
C05410=1106.418,-110.959,-47.034,179.885,4.360,148.748
C05411=1106.413,-110.709,-47.044,179.884,4.365,148.750
C05412=1106.407,-110.458,-47.054,179.884,4.369,148.751
C05413=1106.402,-110.209,-47.063,179.883,4.375,148.752
C05414=1106.397,-109.960,-47.074,179.883,4.380,148.753
C05415=1106.392,-109.710,-47.082,179.883,4.385,148.754
C05416=1106.386,-109.460,-47.093,179.883,4.390,148.756
C05417=1106.381,-109.210,-47.103,179.882,4.394,148.757
C05418=1106.376,-108.961,-47.113,179.881,4.400,148.758
C05419=1106.370,-108.710,-47.122,179.881,4.405,148.760
C05420=1106.365,-108.461,-47.132,179.880,4.410,148.761
C05421=1106.360,-108.211,-47.143,179.880,4.415,148.762
C05422=1106.355,-107.961,-47.153,179.879,4.420,148.763
C05423=1106.350,-107.712,-47.162,179.879,4.425,148.764
C05424=1106.344,-107.462,-47.172,179.879,4.430,148.766
C05425=1106.338,-107.213,-47.182,179.879,4.435,148.767
C05426=1106.334,-106.963,-47.192,179.878,4.440,148.768
C05427=1106.328,-106.712,-47.202,179.878,4.445,148.769
C05428=1106.323,-106.463,-47.212,179.877,4.450,148.770
C05429=1106.318,-106.213,-47.222,179.877,4.455,148.772
C05430=1106.313,-105.963,-47.232,179.876,4.461,148.773
C05431=1106.307,-105.714,-47.242,179.876,4.465,148.774
C05432=1106.302,-105.465,-47.252,179.875,4.470,148.775
C05433=1106.297,-105.214,-47.262,179.875,4.475,148.777
C05434=1106.291,-104.964,-47.272,179.875,4.480,148.778
C05435=1106.286,-104.715,-47.282,179.874,4.485,148.779
C05436=1106.281,-104.465,-47.292,179.874,4.490,148.780
C05437=1106.276,-104.215,-47.302,179.874,4.495,148.781
C05438=1106.270,-103.966,-47.312,179.873,4.500,148.783
C05439=1106.266,-103.716,-47.322,179.873,4.504,148.784
C05440=1106.261,-103.466,-47.333,179.872,4.510,148.785
C05441=1106.255,-103.216,-47.342,179.872,4.515,148.786
C05442=1106.249,-102.966,-47.352,179.872,4.520,148.787
C05443=1106.245,-102.717,-47.362,179.871,4.524,148.789
C05444=1106.239,-102.467,-47.372,179.871,4.529,148.790
C05445=1106.234,-102.217,-47.383,179.870,4.535,148.791
C05446=1106.229,-101.967,-47.393,179.870,4.540,148.792
C05447=1106.224,-101.718,-47.403,179.869,4.544,148.794
C05448=1106.218,-101.468,-47.413,179.869,4.550,148.795
C05449=1106.213,-101.218,-47.424,179.869,4.555,148.796
C05450=1106.208,-100.969,-47.434,179.868,4.559,148.797
C05451=1106.203,-100.754,-47.442,179.868,4.564,148.798
C05452=1106.199,-100.540,-47.451,179.868,4.568,148.799
C05453=1106.194,-100.325,-47.461,179.867,4.572,148.800
C05454=1106.190,-100.110,-47.469,179.867,4.576,148.801
C05455=1106.185,-99.896,-47.477,179.866,4.580,148.802
C05456=1106.180,-99.681,-47.486,179.866,4.585,148.803
C05457=1106.176,-99.467,-47.496,179.866,4.589,148.804
C05458=1106.172,-99.252,-47.504,179.866,4.593,148.805
C05459=1106.166,-99.003,-47.514,179.865,4.598,148.807
C05460=1106.161,-98.752,-47.525,179.865,4.603,148.808
C05461=1106.156,-98.503,-47.535,179.864,4.608,148.809
C05462=1106.150,-98.253,-47.545,179.864,4.613,148.810
C05463=1106.145,-98.003,-47.556,179.864,4.618,148.811
C05464=1106.139,-97.753,-47.566,179.863,4.622,148.813
C05465=1106.135,-97.504,-47.575,179.863,4.628,148.814
C05466=1106.130,-97.254,-47.586,179.863,4.633,148.815
C05467=1106.124,-97.004,-47.596,179.862,4.637,148.816
C05468=1106.119,-96.754,-47.607,179.862,4.642,148.817
C05469=1106.113,-96.505,-47.617,179.861,4.647,148.819
C05470=1106.108,-96.256,-47.628,179.861,4.652,148.820
C05471=1106.103,-96.005,-47.639,179.860,4.657,148.821
C05472=1106.097,-95.756,-47.649,179.860,4.662,148.822
C05473=1106.092,-95.506,-47.659,179.860,4.667,148.823
C05474=1106.087,-95.256,-47.670,179.859,4.671,148.824
C05475=1106.083,-95.006,-47.679,179.859,4.677,148.826
C05476=1106.077,-94.757,-47.690,179.859,4.682,148.827
C05477=1106.071,-94.507,-47.700,179.858,4.686,148.828
C05478=1106.067,-94.258,-47.711,179.858,4.691,148.829
C05479=1106.061,-94.008,-47.721,179.858,4.696,148.830
C05480=1106.056,-93.758,-47.732,179.857,4.701,148.832
C05481=1106.051,-93.508,-47.742,179.857,4.706,148.833
C05482=1106.046,-93.258,-47.753,179.856,4.711,148.834
C05483=1106.040,-93.008,-47.763,179.856,4.715,148.835
C05484=1106.035,-92.759,-47.774,179.855,4.721,148.837
C05485=1106.030,-92.509,-47.784,179.855,4.726,148.838
C05486=1106.024,-92.260,-47.795,179.854,4.730,148.839
C05487=1106.019,-92.009,-47.805,179.854,4.736,148.840
C05488=1106.014,-91.761,-47.816,179.854,4.741,148.841
C05489=1106.009,-91.510,-47.827,179.853,4.745,148.843
C05490=1106.003,-91.261,-47.837,179.853,4.750,148.844
C05491=1105.998,-91.010,-47.848,179.852,4.755,148.845
C05492=1105.993,-90.762,-47.858,179.852,4.760,148.846
C05493=1105.988,-90.511,-47.869,179.851,4.765,148.847
C05494=1105.982,-90.262,-47.879,179.851,4.770,148.849
C05495=1105.977,-90.012,-47.890,179.851,4.775,148.850
C05496=1105.972,-89.763,-47.901,179.851,4.780,148.851
C05497=1105.967,-89.512,-47.911,179.850,4.785,148.852
C05498=1105.961,-89.263,-47.922,179.849,4.790,148.854
C05499=1105.957,-89.013,-47.933,179.849,4.795,148.855
C05500=1105.951,-88.764,-47.943,179.849,4.800,148.856
C05501=1105.946,-88.513,-47.954,179.848,4.805,148.857
C05502=1105.941,-88.264,-47.965,179.848,4.810,148.858
C05503=1105.936,-88.014,-47.975,179.848,4.815,148.859
C05504=1105.930,-87.765,-47.985,179.848,4.820,148.861
C05505=1105.926,-87.515,-47.997,179.847,4.825,148.862
C05506=1105.919,-87.265,-48.007,179.847,4.830,148.863
C05507=1105.916,-87.051,-48.017,179.847,4.835,148.864
C05508=1105.910,-86.836,-48.026,179.846,4.839,148.865
C05509=1105.907,-86.621,-48.035,179.846,4.843,148.866
C05510=1105.902,-86.407,-48.045,179.846,4.848,148.867
C05511=1105.897,-86.193,-48.053,179.846,4.852,148.868
C05512=1105.893,-85.978,-48.063,179.845,4.856,148.869
C05513=1105.888,-85.763,-48.071,179.845,4.860,148.870
C05514=1105.884,-85.549,-48.081,179.845,4.865,148.871
C05515=1105.879,-85.300,-48.092,179.844,4.870,148.873
C05516=1105.874,-85.049,-48.103,179.843,4.875,148.874
C05517=1105.868,-84.800,-48.113,179.843,4.880,148.875
C05518=1105.864,-84.550,-48.124,179.843,4.885,148.876
C05519=1105.857,-84.300,-48.135,179.843,4.890,148.877
C05520=1105.853,-84.051,-48.147,179.843,4.895,148.879
C05521=1105.848,-83.800,-48.157,179.843,4.900,148.880
C05522=1105.842,-83.552,-48.168,179.842,4.906,148.881
C05523=1105.837,-83.301,-48.179,179.842,4.911,148.882
C05524=1105.832,-83.052,-48.190,179.841,4.915,148.884
C05525=1105.826,-82.802,-48.201,179.841,4.921,148.885
C05526=1105.821,-82.553,-48.212,179.841,4.926,148.886
C05527=1105.816,-82.303,-48.222,179.840,4.931,148.887
C05528=1105.811,-82.053,-48.233,179.840,4.936,148.888
C05529=1105.806,-81.803,-48.244,179.840,4.941,148.889
C05530=1105.800,-81.554,-48.256,179.840,4.946,148.891
C05531=1105.795,-81.303,-48.266,179.840,4.951,148.892
C05532=1105.790,-81.054,-48.277,179.840,4.957,148.893
C05533=1105.785,-80.805,-48.288,179.839,4.962,148.894
C05534=1105.779,-80.555,-48.299,179.839,4.967,148.895
C05535=1105.774,-80.305,-48.310,179.839,4.972,148.897
C05536=1105.769,-80.055,-48.321,179.838,4.977,148.898
C05537=1105.764,-79.806,-48.332,179.838,4.982,148.899
C05538=1105.758,-79.556,-48.344,179.838,4.987,148.900
C05539=1105.753,-79.306,-48.354,179.837,4.992,148.902
C05540=1105.748,-79.057,-48.365,179.837,4.997,148.903
C05541=1105.743,-78.807,-48.376,179.837,5.002,148.904
C05542=1105.738,-78.557,-48.388,179.837,5.007,148.905
C05543=1105.732,-78.308,-48.399,179.837,5.013,148.906
C05544=1105.727,-78.058,-48.409,179.837,5.018,148.907
C05545=1105.722,-77.808,-48.421,179.836,5.023,148.909
C05546=1105.717,-77.559,-48.432,179.836,5.028,148.910
C05547=1105.712,-77.309,-48.443,179.836,5.033,148.911
C05548=1105.706,-77.059,-48.455,179.836,5.038,148.912
C05549=1105.701,-76.810,-48.465,179.836,5.043,148.913
C05550=1105.696,-76.560,-48.477,179.836,5.049,148.914
C05551=1105.691,-76.309,-48.488,179.836,5.054,148.916
C05552=1105.685,-76.061,-48.499,179.835,5.059,148.917
C05553=1105.681,-75.811,-48.510,179.835,5.064,148.918
C05554=1105.675,-75.560,-48.521,179.835,5.069,148.919
C05555=1105.670,-75.311,-48.533,179.835,5.074,148.920
C05556=1105.665,-75.062,-48.544,179.835,5.079,148.921
C05557=1105.659,-74.812,-48.555,179.835,5.085,148.923
